LIN {X 0,Y 374.835,Z 474.63,A -85,B 0,C 180,E1 -12336.098,E2 -12336.098} C_VEL
LIN {X 0,Y 375.153,Z 469.967,A -85,B 0,C 180,E1 -12337.535,E2 -12337.535} C_VEL
LIN {X 0,Y 375.66,Z 463.156,A -85,B 0,C 180,E1 -12339.15,E2 -12339.15} C_VEL
LIN {X 0,Y 376.273,Z 455.706,A -85,B 0,C 180,E1 -12340.492,E2 -12340.492} C_VEL
LIN {X 0,Y 376.913,Z 448.357,A -85,B 0,C 180,E1 -12341.563,E2 -12341.563} C_VEL
LIN {X 0,Y 377.501,Z 440.485,A -85,B 0,C 180,E1 -12342.499,E2 -12342.499} C_VEL
LIN {X 0,Y 378.112,Z 432.163,A -85,B 0,C 180,E1 -12343.298,E2 -12343.298} C_VEL
LIN {X 0,Y 378.757,Z 421.529,A -85,B 0,C 180,E1 -12344.095,E2 -12344.095} C_VEL
LIN {X 0,Y 379.284,Z 409.946,A -85,B 0,C 180,E1 -12344.692,E2 -12344.692} C_VEL
LIN {X 0,Y 379.632,Z 400.236,A -85,B 0,C 180,E1 -12345.021,E2 -12345.021} C_VEL
LIN {X 0,Y 380.166,Z 346.091,A -85,B 0,C 180,E1 -12346.072,E2 -12346.072} C_VEL
LIN {X 0,Y 376.584,Z 324.274,A -85,B 0,C 180,E1 -12346.671,E2 -12346.671} C_VEL
LIN {X 0,Y 376.541,Z 323.244,A -85,B 0,C 180,E1 -12346.816,E2 -12346.816} C_VEL
LIN {X 0,Y 377.372,Z 311.444,A -85,B 0,C 180,E1 -12350.153,E2 -12350.153} C_VEL
LIN {X 0,Y 377.425,Z 307.16,A -85,B 0,C 180,E1 -12351.402,E2 -12351.402} C_VEL
LIN {X 0,Y 376.03,Z 298.57,A -85,B 0,C 180,E1 -12354.068,E2 -12354.068} C_VEL
LIN {X 0,Y 375.922,Z 298.47,A -85,B 0,C 180,E1 -12357.864,E2 -12357.864} C_VEL
LIN {X 0,Y 375.953,Z 298.469,A -85,B 0,C 180,E1 -12361.562,E2 -12361.562} C_VEL
LIN {X 0,Y 375.951,Z 298.47,A -85,B 0,C 180,E1 -12365.415,E2 -12365.415} C_VEL
LIN {X 0,Y 375.931,Z 298.466,A -85,B 0,C 180,E1 -12368.262,E2 -12368.262} C_VEL
LIN {X 0,Y 375.908,Z 298.472,A -85,B 0,C 180,E1 -12371.596,E2 -12371.596} C_VEL
LIN {X 0,Y 375.915,Z 298.471,A -85,B 0,C 180,E1 -12374.73,E2 -12374.73} C_VEL
LIN {X 0,Y 375.901,Z 298.471,A -85,B 0,C 180,E1 -12377.696,E2 -12377.696} C_VEL
LIN {X 0,Y 375.928,Z 298.469,A -85,B 0,C 180,E1 -12380.533,E2 -12380.533} C_VEL
LIN {X 0,Y 375.951,Z 298.465,A -85,B 0,C 180,E1 -12383.496,E2 -12383.496} C_VEL
LIN {X 0,Y 375.95,Z 298.464,A -85,B 0,C 180,E1 -12385.888,E2 -12385.888} C_VEL
LIN {X 0,Y 375.953,Z 298.464,A -85,B 0,C 180,E1 -12389.686,E2 -12389.686} C_VEL
LIN {X 0,Y 375.909,Z 298.47,A -85,B 0,C 180,E1 -12392.134,E2 -12392.134} C_VEL
LIN {X 0,Y 375.928,Z 298.472,A -85,B 0,C 180,E1 -12394.533,E2 -12394.533} C_VEL
LIN {X 0,Y 375.962,Z 298.466,A -85,B 0,C 180,E1 -12396.886,E2 -12396.886} C_VEL
LIN {X 0,Y 375.965,Z 298.467,A -85,B 0,C 180,E1 -12400.338,E2 -12400.338} C_VEL
LIN {X 0,Y 375.964,Z 298.463,A -85,B 0,C 180,E1 -12403.716,E2 -12403.716} C_VEL
LIN {X 0,Y 376.094,Z 298.447,A -85,B 0,C 180,E1 -12407.042,E2 -12407.042} C_VEL
LIN {X 0,Y 376.103,Z 298.451,A -85,B 0,C 180,E1 -12410.318,E2 -12410.318} C_VEL
LIN {X 0,Y 376.188,Z 298.435,A -85,B 0,C 180,E1 -12413.564,E2 -12413.564} C_VEL
LIN {X 0,Y 376.327,Z 298.421,A -85,B 0,C 180,E1 -12417.86,E2 -12417.86} C_VEL
LIN {X 0,Y 376.322,Z 298.422,A -85,B 0,C 180,E1 -12422.141,E2 -12422.141} C_VEL
LIN {X 0,Y 376.188,Z 298.436,A -85,B 0,C 180,E1 -12426.436,E2 -12426.436} C_VEL
LIN {X 0,Y 376.097,Z 298.451,A -85,B 0,C 180,E1 -12429.682,E2 -12429.682} C_VEL
LIN {X 0,Y 376.081,Z 298.454,A -85,B 0,C 180,E1 -12433.658,E2 -12433.658} C_VEL
LIN {X 0,Y 375.998,Z 298.465,A -85,B 0,C 180,E1 -12437.589,E2 -12437.589} C_VEL
LIN {X 0,Y 375.971,Z 298.462,A -85,B 0,C 180,E1 -12440.833,E2 -12440.833} C_VEL
LIN {X 0,Y 375.926,Z 298.467,A -85,B 0,C 180,E1 -12444.286,E2 -12444.286} C_VEL
LIN {X 0,Y 375.903,Z 298.47,A -85,B 0,C 180,E1 -12446.661,E2 -12446.661} C_VEL
LIN {X 0,Y 375.906,Z 298.473,A -85,B 0,C 180,E1 -12449.085,E2 -12449.085} C_VEL
LIN {X 0,Y 375.947,Z 298.467,A -85,B 0,C 180,E1 -12451.563,E2 -12451.563} C_VEL
LIN {X 0,Y 375.943,Z 298.469,A -85,B 0,C 180,E1 -12455.417,E2 -12455.417} C_VEL
LIN {X 0,Y 375.929,Z 298.467,A -85,B 0,C 180,E1 -12458.263,E2 -12458.263} C_VEL
LIN {X 0,Y 375.908,Z 298.47,A -85,B 0,C 180,E1 -12461.598,E2 -12461.598} C_VEL
LIN {X 0,Y 375.916,Z 298.472,A -85,B 0,C 180,E1 -12464.731,E2 -12464.731} C_VEL
LIN {X 0,Y 375.903,Z 298.47,A -85,B 0,C 180,E1 -12467.697,E2 -12467.697} C_VEL
LIN {X 0,Y 375.931,Z 298.47,A -85,B 0,C 180,E1 -12470.535,E2 -12470.535} C_VEL
LIN {X 0,Y 375.959,Z 298.463,A -85,B 0,C 180,E1 -12473.497,E2 -12473.497} C_VEL
LIN {X 0,Y 375.956,Z 298.464,A -85,B 0,C 180,E1 -12475.889,E2 -12475.889} C_VEL
LIN {X 0,Y 375.957,Z 298.463,A -85,B 0,C 180,E1 -12479.688,E2 -12479.688} C_VEL
LIN {X 0,Y 375.915,Z 298.471,A -85,B 0,C 180,E1 -12482.136,E2 -12482.136} C_VEL
LIN {X 0,Y 376.046,Z 298.57,A -85,B 0,C 180,E1 -12485.976,E2 -12485.976} C_VEL
LIN {X 0,Y 377.411,Z 307.03,A -85,B 0,C 180,E1 -12488.604,E2 -12488.604} C_VEL
LIN {X 0,Y 377.223,Z 313.241,A -85,B 0,C 180,E1 -12490.406,E2 -12490.406} C_VEL
LIN {X 0,Y 376.539,Z 323.725,A -85,B 0,C 180,E1 -12493.324,E2 -12493.324} C_VEL
LIN {X 0,Y 377.181,Z 328.108,A -85,B 0,C 180,E1 -12493.493,E2 -12493.493} C_VEL
LIN {X 0,Y 380.2,Z 346.979,A -85,B 0,C 180,E1 -12493.992,E2 -12493.992} C_VEL
LIN {X 0,Y 379.651,Z 399.832,A -85,B 0,C 180,E1 -12495.014,E2 -12495.014} C_VEL
LIN {X 0,Y 379.356,Z 408.855,A -85,B 0,C 180,E1 -12495.311,E2 -12495.311} C_VEL
LIN {X 0,Y 378.925,Z 418.416,A -85,B 0,C 180,E1 -12495.774,E2 -12495.774} C_VEL
LIN {X 0,Y 378.378,Z 428.445,A -85,B 0,C 180,E1 -12496.438,E2 -12496.438} C_VEL
LIN {X 0,Y 377.632,Z 438.849,A -85,B 0,C 180,E1 -12497.369,E2 -12497.369} C_VEL
LIN {X 0,Y 377.021,Z 446.999,A -85,B 0,C 180,E1 -12498.304,E2 -12498.304} C_VEL
LIN {X 0,Y 376.473,Z 453.724,A -85,B 0,C 180,E1 -12499.241,E2 -12499.241} C_VEL
LIN {X 0,Y 375.895,Z 460.092,A -85,B 0,C 180,E1 -12500.313,E2 -12500.313} C_VEL
LIN {X 0,Y 375.406,Z 466.559,A -85,B 0,C 180,E1 -12501.658,E2 -12501.658} C_VEL
LIN {X 0,Y 375.086,Z 471.723,A -85,B 0,C 180,E1 -12503.005,E2 -12503.005} C_VEL
LIN {X 0,Y 374.779,Z 476.499,A -85,B 0,C 180,E1 -12504.62,E2 -12504.62} C_VEL
LIN {X 0,Y 374.64,Z 478.829,A -85,B 0,C 180,E1 -12505.697,E2 -12505.697} C_VEL
LIN {X 0,Y 374.492,Z 480.603,A -85,B 0,C 180,E1 -12506.773,E2 -12506.773} C_VEL
LIN {X 0,Y 374.461,Z 481.882,A -85,B 0,C 180,E1 -12507.849,E2 -12507.849} C_VEL
LIN {X 0,Y 374.457,Z 482.69,A -85,B 0,C 180,E1 -12508.925,E2 -12508.925} C_VEL
LIN {X 0,Y 374.44,Z 482.998,A -85,B 0,C 180,E1 -12510,E2 -12510} C_VEL
LIN {X 0,Y 374.454,Z 482.72,A -85,B 0,C 180,E1 -12511.075,E2 -12511.075} C_VEL
LIN {X 0,Y 374.444,Z 481.973,A -85,B 0,C 180,E1 -12512.151,E2 -12512.151} C_VEL
LIN {X 0,Y 374.485,Z 480.755,A -85,B 0,C 180,E1 -12513.227,E2 -12513.227} C_VEL
LIN {X 0,Y 374.707,Z 477.894,A -85,B 0,C 180,E1 -12514.842,E2 -12514.842} C_VEL
LIN {X 0,Y 374.825,Z 474.83,A -85,B 0,C 180,E1 -12516.083,E2 -12516.083} C_VEL
LIN {X 0,Y 375.16,Z 470.167,A -85,B 0,C 180,E1 -12517.535,E2 -12517.535} C_VEL
LIN {X 0,Y 375.545,Z 464.655,A -85,B 0,C 180,E1 -12518.881,E2 -12518.881} C_VEL
LIN {X 0,Y 376.175,Z 457.735,A -85,B 0,C 180,E1 -12520.223,E2 -12520.223} C_VEL
LIN {X 0,Y 376.798,Z 449.79,A -85,B 0,C 180,E1 -12521.43,E2 -12521.43} C_VEL
LIN {X 0,Y 377.376,Z 442.216,A -85,B 0,C 180,E1 -12522.366,E2 -12522.366} C_VEL
LIN {X 0,Y 378.043,Z 434.279,A -85,B 0,C 180,E1 -12523.163,E2 -12523.163} C_VEL
LIN {X 0,Y 378.538,Z 426.084,A -85,B 0,C 180,E1 -12523.83,E2 -12523.83} C_VEL
LIN {X 0,Y 378.982,Z 417.782,A -85,B 0,C 180,E1 -12524.361,E2 -12524.361} C_VEL
LIN {X 0,Y 379.342,Z 408.815,A -85,B 0,C 180,E1 -12524.792,E2 -12524.792} C_VEL
LIN {X 0,Y 379.53,Z 403.476,A -85,B 0,C 180,E1 -12524.995,E2 -12524.995} C_VEL
LIN {X 0,Y 379.115,Z 397.696,A -85,B 0,C 180,E1 -12525.169,E2 -12525.169} C_VEL
LIN {X 0,Y 376.426,Z 388.36,A -85,B 0,C 180,E1 -12525.475,E2 -12525.475} C_VEL
LIN {X 0,Y 373.709,Z 379.004,A -85,B 0,C 180,E1 -12525.772,E2 -12525.772} C_VEL
LIN {X 0,Y 373.119,Z 373.187,A -85,B 0,C 180,E1 -12525.909,E2 -12525.909} C_VEL
LIN {X 0,Y 373.222,Z 346.278,A -85,B 0,C 180,E1 -12526.433,E2 -12526.433} C_VEL
LIN {X 0,Y 369.609,Z 324.06,A -85,B 0,C 180,E1 -12527.07,E2 -12527.07} C_VEL
LIN {X 0,Y 369.646,Z 322.378,A -85,B 0,C 180,E1 -12527.424,E2 -12527.424} C_VEL
LIN {X 0,Y 370.417,Z 311.641,A -85,B 0,C 180,E1 -12530.548,E2 -12530.548} C_VEL
LIN {X 0,Y 370.302,Z 307.197,A -85,B 0,C 180,E1 -12531.882,E2 -12531.882} C_VEL
LIN {X 0,Y 368.991,Z 299.445,A -85,B 0,C 180,E1 -12534.36,E2 -12534.36} C_VEL
LIN {X 0,Y 368.863,Z 299.349,A -85,B 0,C 180,E1 -12537.211,E2 -12537.211} C_VEL
LIN {X 0,Y 368.892,Z 299.348,A -85,B 0,C 180,E1 -12539.692,E2 -12539.692} C_VEL
LIN {X 0,Y 368.894,Z 299.345,A -85,B 0,C 180,E1 -12543.042,E2 -12543.042} C_VEL
LIN {X 0,Y 368.913,Z 299.341,A -85,B 0,C 180,E1 -12546.196,E2 -12546.196} C_VEL
LIN {X 0,Y 368.871,Z 299.349,A -85,B 0,C 180,E1 -12548.956,E2 -12548.956} C_VEL
LIN {X 0,Y 368.854,Z 299.348,A -85,B 0,C 180,E1 -12552.004,E2 -12552.004} C_VEL
LIN {X 0,Y 368.869,Z 299.352,A -85,B 0,C 180,E1 -12555.174,E2 -12555.174} C_VEL
LIN {X 0,Y 368.859,Z 299.347,A -85,B 0,C 180,E1 -12558.174,E2 -12558.174} C_VEL
LIN {X 0,Y 368.872,Z 299.348,A -85,B 0,C 180,E1 -12561.365,E2 -12561.365} C_VEL
LIN {X 0,Y 368.925,Z 299.343,A -85,B 0,C 180,E1 -12565.145,E2 -12565.145} C_VEL
LIN {X 0,Y 368.906,Z 299.345,A -85,B 0,C 180,E1 -12569.044,E2 -12569.044} C_VEL
LIN {X 0,Y 368.9,Z 299.342,A -85,B 0,C 180,E1 -12571.557,E2 -12571.557} C_VEL
LIN {X 0,Y 368.878,Z 299.346,A -85,B 0,C 180,E1 -12575.219,E2 -12575.219} C_VEL
LIN {X 0,Y 368.888,Z 299.344,A -85,B 0,C 180,E1 -12577.602,E2 -12577.602} C_VEL
LIN {X 0,Y 368.905,Z 299.343,A -85,B 0,C 180,E1 -12581.103,E2 -12581.103} C_VEL
LIN {X 0,Y 368.93,Z 299.344,A -85,B 0,C 180,E1 -12584.532,E2 -12584.532} C_VEL
LIN {X 0,Y 369.049,Z 299.326,A -85,B 0,C 180,E1 -12586.79,E2 -12586.79} C_VEL
LIN {X 0,Y 369.054,Z 299.328,A -85,B 0,C 180,E1 -12590.131,E2 -12590.131} C_VEL
LIN {X 0,Y 369.149,Z 299.312,A -85,B 0,C 180,E1 -12593.441,E2 -12593.441} C_VEL
LIN {X 0,Y 369.291,Z 299.297,A -85,B 0,C 180,E1 -12597.819,E2 -12597.819} C_VEL
LIN {X 0,Y 369.285,Z 299.298,A -85,B 0,C 180,E1 -12602.181,E2 -12602.181} C_VEL
LIN {X 0,Y 369.148,Z 299.312,A -85,B 0,C 180,E1 -12606.559,E2 -12606.559} C_VEL
LIN {X 0,Y 369.048,Z 299.329,A -85,B 0,C 180,E1 -12609.869,E2 -12609.869} C_VEL
LIN {X 0,Y 369.029,Z 299.332,A -85,B 0,C 180,E1 -12613.772,E2 -12613.772} C_VEL
LIN {X 0,Y 368.945,Z 299.341,A -85,B 0,C 180,E1 -12617.745,E2 -12617.745} C_VEL
LIN {X 0,Y 368.901,Z 299.346,A -85,B 0,C 180,E1 -12621.221,E2 -12621.221} C_VEL
LIN {X 0,Y 368.899,Z 299.344,A -85,B 0,C 180,E1 -12623.874,E2 -12623.874} C_VEL
LIN {X 0,Y 368.849,Z 299.354,A -85,B 0,C 180,E1 -12627.212,E2 -12627.212} C_VEL
LIN {X 0,Y 368.885,Z 299.346,A -85,B 0,C 180,E1 -12629.693,E2 -12629.693} C_VEL
LIN {X 0,Y 368.889,Z 299.348,A -85,B 0,C 180,E1 -12633.043,E2 -12633.043} C_VEL
LIN {X 0,Y 368.904,Z 299.342,A -85,B 0,C 180,E1 -12636.198,E2 -12636.198} C_VEL
LIN {X 0,Y 368.867,Z 299.352,A -85,B 0,C 180,E1 -12638.958,E2 -12638.958} C_VEL
LIN {X 0,Y 368.852,Z 299.348,A -85,B 0,C 180,E1 -12642.006,E2 -12642.006} C_VEL
LIN {X 0,Y 368.868,Z 299.35,A -85,B 0,C 180,E1 -12645.175,E2 -12645.175} C_VEL
LIN {X 0,Y 368.855,Z 299.349,A -85,B 0,C 180,E1 -12648.175,E2 -12648.175} C_VEL
LIN {X 0,Y 368.871,Z 299.347,A -85,B 0,C 180,E1 -12651.367,E2 -12651.367} C_VEL
LIN {X 0,Y 368.931,Z 299.34,A -85,B 0,C 180,E1 -12655.147,E2 -12655.147} C_VEL
LIN {X 0,Y 368.91,Z 299.343,A -85,B 0,C 180,E1 -12659.045,E2 -12659.045} C_VEL
LIN {X 0,Y 368.904,Z 299.342,A -85,B 0,C 180,E1 -12661.558,E2 -12661.558} C_VEL
LIN {X 0,Y 368.937,Z 299.34,A -85,B 0,C 180,E1 -12665.224,E2 -12665.224} C_VEL
LIN {X 0,Y 368.964,Z 299.455,A -85,B 0,C 180,E1 -12665.699,E2 -12665.699} C_VEL
LIN {X 0,Y 370.297,Z 307.05,A -85,B 0,C 180,E1 -12668.118,E2 -12668.118} C_VEL
LIN {X 0,Y 370.438,Z 311.49,A -85,B 0,C 180,E1 -12669.453,E2 -12669.453} C_VEL
LIN {X 0,Y 369.575,Z 323.615,A -85,B 0,C 180,E1 -12672.929,E2 -12672.929} C_VEL
LIN {X 0,Y 370.085,Z 326.931,A -85,B 0,C 180,E1 -12673.085,E2 -12673.085} C_VEL
LIN {X 0,Y 373.379,Z 347.391,A -85,B 0,C 180,E1 -12673.641,E2 -12673.641} C_VEL
LIN {X 0,Y 372.867,Z 399.709,A -85,B 0,C 180,E1 -12674.674,E2 -12674.674} C_VEL
LIN {X 0,Y 372.455,Z 409.396,A -85,B 0,C 180,E1 -12674.998,E2 -12674.998} C_VEL
LIN {X 0,Y 372.037,Z 419.413,A -85,B 0,C 180,E1 -12675.505,E2 -12675.505} C_VEL
LIN {X 0,Y 371.299,Z 430.789,A -85,B 0,C 180,E1 -12676.314,E2 -12676.314} C_VEL
LIN {X 0,Y 370.649,Z 439.356,A -85,B 0,C 180,E1 -12677.127,E2 -12677.127} C_VEL
LIN {X 0,Y 370.052,Z 447.415,A -85,B 0,C 180,E1 -12678.081,E2 -12678.081} C_VEL
LIN {X 0,Y 369.467,Z 454.071,A -85,B 0,C 180,E1 -12679.035,E2 -12679.035} C_VEL
LIN {X 0,Y 368.886,Z 460.388,A -85,B 0,C 180,E1 -12680.127,E2 -12680.127} C_VEL
LIN {X 0,Y 368.433,Z 465.635,A -85,B 0,C 180,E1 -12681.222,E2 -12681.222} C_VEL
LIN {X 0,Y 368.124,Z 470.009,A -85,B 0,C 180,E1 -12682.32,E2 -12682.32} C_VEL
LIN {X 0,Y 367.734,Z 475.123,A -85,B 0,C 180,E1 -12683.951,E2 -12683.951} C_VEL
LIN {X 0,Y 367.64,Z 477.799,A -85,B 0,C 180,E1 -12685.065,E2 -12685.065} C_VEL
LIN {X 0,Y 367.41,Z 480.688,A -85,B 0,C 180,E1 -12686.71,E2 -12686.71} C_VEL
LIN {X 0,Y 367.362,Z 481.933,A -85,B 0,C 180,E1 -12687.807,E2 -12687.807} C_VEL
LIN {X 0,Y 367.355,Z 482.707,A -85,B 0,C 180,E1 -12688.904,E2 -12688.904} C_VEL
LIN {X 0,Y 367.34,Z 483,A -85,B 0,C 180,E1 -12690,E2 -12690} C_VEL
LIN {X 0,Y 367.355,Z 482.704,A -85,B 0,C 180,E1 -12691.096,E2 -12691.096} C_VEL
LIN {X 0,Y 367.362,Z 481.922,A -85,B 0,C 180,E1 -12692.193,E2 -12692.193} C_VEL
LIN {X 0,Y 367.41,Z 480.67,A -85,B 0,C 180,E1 -12693.29,E2 -12693.29} C_VEL
LIN {X 0,Y 367.633,Z 477.774,A -85,B 0,C 180,E1 -12694.935,E2 -12694.935} C_VEL
LIN {X 0,Y 367.836,Z 473.783,A -85,B 0,C 180,E1 -12696.522,E2 -12696.522} C_VEL
LIN {X 0,Y 368.253,Z 467.925,A -85,B 0,C 180,E1 -12698.229,E2 -12698.229} C_VEL
LIN {X 0,Y 368.767,Z 461.741,A -85,B 0,C 180,E1 -12699.599,E2 -12699.599} C_VEL
LIN {X 0,Y 369.29,Z 455.704,A -85,B 0,C 180,E1 -12700.693,E2 -12700.693} C_VEL
LIN {X 0,Y 369.966,Z 448.354,A -85,B 0,C 180,E1 -12701.783,E2 -12701.783} C_VEL
LIN {X 0,Y 370.567,Z 440.481,A -85,B 0,C 180,E1 -12702.737,E2 -12702.737} C_VEL
LIN {X 0,Y 371.208,Z 432.159,A -85,B 0,C 180,E1 -12703.55,E2 -12703.55} C_VEL
LIN {X 0,Y 371.888,Z 421.524,A -85,B 0,C 180,E1 -12704.361,E2 -12704.361} C_VEL
LIN {X 0,Y 372.437,Z 409.937,A -85,B 0,C 180,E1 -12704.968,E2 -12704.968} C_VEL
LIN {X 0,Y 372.791,Z 400.221,A -85,B 0,C 180,E1 -12705.303,E2 -12705.303} C_VEL
LIN {X 0,Y 373.377,Z 346.955,A -85,B 0,C 180,E1 -12706.355,E2 -12706.355} C_VEL
LIN {X 0,Y 369.632,Z 324.261,A -85,B 0,C 180,E1 -12706.994,E2 -12706.994} C_VEL
LIN {X 0,Y 369.572,Z 323.242,A -85,B 0,C 180,E1 -12707.143,E2 -12707.143} C_VEL
LIN {X 0,Y 370.422,Z 311.442,A -85,B 0,C 180,E1 -12710.548,E2 -12710.548} C_VEL
LIN {X 0,Y 370.291,Z 307.003,A -85,B 0,C 180,E1 -12711.882,E2 -12711.882} C_VEL
LIN {X 0,Y 368.982,Z 299.443,A -85,B 0,C 180,E1 -12714.297,E2 -12714.297} C_VEL
LIN {X 0,Y 368.861,Z 299.35,A -85,B 0,C 180,E1 -12717.211,E2 -12717.211} C_VEL
LIN {X 0,Y 368.891,Z 299.348,A -85,B 0,C 180,E1 -12719.692,E2 -12719.692} C_VEL
LIN {X 0,Y 368.892,Z 299.346,A -85,B 0,C 180,E1 -12723.042,E2 -12723.042} C_VEL
LIN {X 0,Y 368.911,Z 299.341,A -85,B 0,C 180,E1 -12726.196,E2 -12726.196} C_VEL
LIN {X 0,Y 368.869,Z 299.349,A -85,B 0,C 180,E1 -12728.956,E2 -12728.956} C_VEL
LIN {X 0,Y 368.853,Z 299.348,A -85,B 0,C 180,E1 -12732.005,E2 -12732.005} C_VEL
LIN {X 0,Y 368.868,Z 299.352,A -85,B 0,C 180,E1 -12735.174,E2 -12735.174} C_VEL
LIN {X 0,Y 368.854,Z 299.348,A -85,B 0,C 180,E1 -12738.174,E2 -12738.174} C_VEL
LIN {X 0,Y 368.87,Z 299.348,A -85,B 0,C 180,E1 -12741.366,E2 -12741.366} C_VEL
LIN {X 0,Y 368.924,Z 299.343,A -85,B 0,C 180,E1 -12745.145,E2 -12745.145} C_VEL
LIN {X 0,Y 368.906,Z 299.345,A -85,B 0,C 180,E1 -12749.044,E2 -12749.044} C_VEL
LIN {X 0,Y 368.899,Z 299.342,A -85,B 0,C 180,E1 -12751.557,E2 -12751.557} C_VEL
LIN {X 0,Y 368.877,Z 299.346,A -85,B 0,C 180,E1 -12755.219,E2 -12755.219} C_VEL
LIN {X 0,Y 368.888,Z 299.344,A -85,B 0,C 180,E1 -12757.602,E2 -12757.602} C_VEL
LIN {X 0,Y 368.905,Z 299.343,A -85,B 0,C 180,E1 -12761.103,E2 -12761.103} C_VEL
LIN {X 0,Y 368.93,Z 299.343,A -85,B 0,C 180,E1 -12764.532,E2 -12764.532} C_VEL
LIN {X 0,Y 369.049,Z 299.326,A -85,B 0,C 180,E1 -12766.79,E2 -12766.79} C_VEL
LIN {X 0,Y 369.053,Z 299.328,A -85,B 0,C 180,E1 -12770.131,E2 -12770.131} C_VEL
LIN {X 0,Y 369.149,Z 299.312,A -85,B 0,C 180,E1 -12773.441,E2 -12773.441} C_VEL
LIN {X 0,Y 369.291,Z 299.297,A -85,B 0,C 180,E1 -12777.819,E2 -12777.819} C_VEL
LIN {X 0,Y 369.285,Z 299.298,A -85,B 0,C 180,E1 -12782.181,E2 -12782.181} C_VEL
LIN {X 0,Y 369.149,Z 299.312,A -85,B 0,C 180,E1 -12786.559,E2 -12786.559} C_VEL
LIN {X 0,Y 369.048,Z 299.329,A -85,B 0,C 180,E1 -12789.869,E2 -12789.869} C_VEL
LIN {X 0,Y 369.029,Z 299.332,A -85,B 0,C 180,E1 -12793.772,E2 -12793.772} C_VEL
LIN {X 0,Y 368.945,Z 299.341,A -85,B 0,C 180,E1 -12797.745,E2 -12797.745} C_VEL
LIN {X 0,Y 368.901,Z 299.345,A -85,B 0,C 180,E1 -12801.221,E2 -12801.221} C_VEL
LIN {X 0,Y 368.9,Z 299.344,A -85,B 0,C 180,E1 -12803.874,E2 -12803.874} C_VEL
LIN {X 0,Y 368.85,Z 299.353,A -85,B 0,C 180,E1 -12807.213,E2 -12807.213} C_VEL
LIN {X 0,Y 368.885,Z 299.346,A -85,B 0,C 180,E1 -12809.693,E2 -12809.693} C_VEL
LIN {X 0,Y 368.889,Z 299.348,A -85,B 0,C 180,E1 -12813.043,E2 -12813.043} C_VEL
LIN {X 0,Y 368.905,Z 299.342,A -85,B 0,C 180,E1 -12816.198,E2 -12816.198} C_VEL
LIN {X 0,Y 368.868,Z 299.351,A -85,B 0,C 180,E1 -12818.958,E2 -12818.958} C_VEL
LIN {X 0,Y 368.853,Z 299.348,A -85,B 0,C 180,E1 -12822.006,E2 -12822.006} C_VEL
LIN {X 0,Y 368.869,Z 299.35,A -85,B 0,C 180,E1 -12825.175,E2 -12825.175} C_VEL
LIN {X 0,Y 368.856,Z 299.348,A -85,B 0,C 180,E1 -12828.175,E2 -12828.175} C_VEL
LIN {X 0,Y 368.873,Z 299.347,A -85,B 0,C 180,E1 -12831.367,E2 -12831.367} C_VEL
LIN {X 0,Y 368.933,Z 299.34,A -85,B 0,C 180,E1 -12835.147,E2 -12835.147} C_VEL
LIN {X 0,Y 368.894,Z 299.345,A -85,B 0,C 180,E1 -12839.044,E2 -12839.044} C_VEL
LIN {X 0,Y 368.905,Z 299.342,A -85,B 0,C 180,E1 -12841.558,E2 -12841.558} C_VEL
LIN {X 0,Y 368.935,Z 299.342,A -85,B 0,C 180,E1 -12845.224,E2 -12845.224} C_VEL
LIN {X 0,Y 369.008,Z 299.593,A -85,B 0,C 180,E1 -12845.826,E2 -12845.826} C_VEL
LIN {X 0,Y 370.38,Z 307.778,A -85,B 0,C 180,E1 -12848.401,E2 -12848.401} C_VEL
LIN {X 0,Y 370.311,Z 313.243,A -85,B 0,C 180,E1 -12850.025,E2 -12850.025} C_VEL
LIN {X 0,Y 369.576,Z 323.586,A -85,B 0,C 180,E1 -12852.975,E2 -12852.975} C_VEL
LIN {X 0,Y 369.703,Z 324.949,A -85,B 0,C 180,E1 -12853.077,E2 -12853.077} C_VEL
LIN {X 0,Y 373.378,Z 347.27,A -85,B 0,C 180,E1 -12853.696,E2 -12853.696} C_VEL
LIN {X 0,Y 372.808,Z 399.85,A -85,B 0,C 180,E1 -12854.732,E2 -12854.732} C_VEL
LIN {X 0,Y 372.506,Z 408.867,A -85,B 0,C 180,E1 -12855.035,E2 -12855.035} C_VEL
LIN {X 0,Y 372.064,Z 418.425,A -85,B 0,C 180,E1 -12855.506,E2 -12855.506} C_VEL
LIN {X 0,Y 371.49,Z 428.452,A -85,B 0,C 180,E1 -12856.182,E2 -12856.182} C_VEL
LIN {X 0,Y 370.7,Z 438.854,A -85,B 0,C 180,E1 -12857.129,E2 -12857.129} C_VEL
LIN {X 0,Y 370.068,Z 447.003,A -85,B 0,C 180,E1 -12858.081,E2 -12858.081} C_VEL
LIN {X 0,Y 369.486,Z 453.727,A -85,B 0,C 180,E1 -12859.035,E2 -12859.035} C_VEL
LIN {X 0,Y 368.895,Z 460.094,A -85,B 0,C 180,E1 -12860.127,E2 -12860.127} C_VEL
LIN {X 0,Y 368.385,Z 466.562,A -85,B 0,C 180,E1 -12861.498,E2 -12861.498} C_VEL
LIN {X 0,Y 368.041,Z 471.722,A -85,B 0,C 180,E1 -12862.87,E2 -12862.87} C_VEL
LIN {X 0,Y 367.688,Z 476.5,A -85,B 0,C 180,E1 -12864.516,E2 -12864.516} C_VEL
LIN {X 0,Y 367.577,Z 478.83,A -85,B 0,C 180,E1 -12865.614,E2 -12865.614} C_VEL
LIN {X 0,Y 367.412,Z 480.604,A -85,B 0,C 180,E1 -12866.71,E2 -12866.71} C_VEL
LIN {X 0,Y 367.363,Z 481.883,A -85,B 0,C 180,E1 -12867.807,E2 -12867.807} C_VEL
LIN {X 0,Y 367.356,Z 482.69,A -85,B 0,C 180,E1 -12868.904,E2 -12868.904} C_VEL
LIN {X 0,Y 367.341,Z 482.998,A -85,B 0,C 180,E1 -12870,E2 -12870} C_VEL
LIN {X 0,Y 367.353,Z 482.72,A -85,B 0,C 180,E1 -12871.096,E2 -12871.096} C_VEL
LIN {X 0,Y 367.347,Z 481.973,A -85,B 0,C 180,E1 -12872.193,E2 -12872.193} C_VEL
LIN {X 0,Y 367.405,Z 480.755,A -85,B 0,C 180,E1 -12873.29,E2 -12873.29} C_VEL
LIN {X 0,Y 367.629,Z 477.893,A -85,B 0,C 180,E1 -12874.935,E2 -12874.935} C_VEL
LIN {X 0,Y 367.831,Z 473.962,A -85,B 0,C 180,E1 -12876.514,E2 -12876.514} C_VEL
LIN {X 0,Y 368.247,Z 468.168,A -85,B 0,C 180,E1 -12878.229,E2 -12878.229} C_VEL
LIN {X 0,Y 368.767,Z 462.037,A -85,B 0,C 180,E1 -12879.599,E2 -12879.599} C_VEL
LIN {X 0,Y 369.301,Z 456.051,A -85,B 0,C 180,E1 -12880.693,E2 -12880.693} C_VEL
LIN {X 0,Y 369.914,Z 448.766,A -85,B 0,C 180,E1 -12881.785,E2 -12881.785} C_VEL
LIN {X 0,Y 370.52,Z 440.982,A -85,B 0,C 180,E1 -12882.738,E2 -12882.738} C_VEL
LIN {X 0,Y 371.239,Z 432.773,A -85,B 0,C 180,E1 -12883.548,E2 -12883.548} C_VEL
LIN {X 0,Y 371.775,Z 424.204,A -85,B 0,C 180,E1 -12884.226,E2 -12884.226} C_VEL
LIN {X 0,Y 372.372,Z 412.86,A -85,B 0,C 180,E1 -12884.901,E2 -12884.901} C_VEL
LIN {X 0,Y 372.762,Z 401.287,A -85,B 0,C 180,E1 -12885.333,E2 -12885.333} C_VEL
LIN {X 0,Y 373.119,Z 373.187,A -85,B 0,C 180,E1 -12885.909,E2 -12885.909} C_VEL
LIN {X 0,Y 372.608,Z 367.369,A -85,B 0,C 180,E1 -12886.046,E2 -12886.046} C_VEL
LIN {X 0,Y 370.067,Z 357.998,A -85,B 0,C 180,E1 -12886.344,E2 -12886.344} C_VEL
LIN {X 0,Y 366.559,Z 346.793,A -85,B 0,C 180,E1 -12886.729,E2 -12886.729} C_VEL
LIN {X 0,Y 365.808,Z 342.941,A -85,B 0,C 180,E1 -12886.842,E2 -12886.842} C_VEL
LIN {X 0,Y 362.669,Z 324.052,A -85,B 0,C 180,E1 -12887.407,E2 -12887.407} C_VEL
LIN {X 0,Y 362.693,Z 322.376,A -85,B 0,C 180,E1 -12887.769,E2 -12887.769} C_VEL
LIN {X 0,Y 363.472,Z 311.639,A -85,B 0,C 180,E1 -12890.959,E2 -12890.959} C_VEL
LIN {X 0,Y 363.19,Z 307.567,A -85,B 0,C 180,E1 -12892.22,E2 -12892.22} C_VEL
LIN {X 0,Y 361.939,Z 300.324,A -85,B 0,C 180,E1 -12894.59,E2 -12894.59} C_VEL
LIN {X 0,Y 361.838,Z 300.226,A -85,B 0,C 180,E1 -12897.784,E2 -12897.784} C_VEL
LIN {X 0,Y 361.845,Z 300.225,A -85,B 0,C 180,E1 -12901.285,E2 -12901.285} C_VEL
LIN {X 0,Y 361.851,Z 300.22,A -85,B 0,C 180,E1 -12904.28,E2 -12904.28} C_VEL
LIN {X 0,Y 361.857,Z 300.225,A -85,B 0,C 180,E1 -12907.221,E2 -12907.221} C_VEL
LIN {X 0,Y 361.806,Z 300.227,A -85,B 0,C 180,E1 -12910.75,E2 -12910.75} C_VEL
LIN {X 0,Y 361.807,Z 300.226,A -85,B 0,C 180,E1 -12914.369,E2 -12914.369} C_VEL
LIN {X 0,Y 361.821,Z 300.226,A -85,B 0,C 180,E1 -12917.569,E2 -12917.569} C_VEL
LIN {X 0,Y 361.838,Z 300.223,A -85,B 0,C 180,E1 -12921.571,E2 -12921.571} C_VEL
LIN {X 0,Y 361.864,Z 300.222,A -85,B 0,C 180,E1 -12924.656,E2 -12924.656} C_VEL
LIN {X 0,Y 361.831,Z 300.225,A -85,B 0,C 180,E1 -12928.37,E2 -12928.37} C_VEL
LIN {X 0,Y 361.86,Z 300.223,A -85,B 0,C 180,E1 -12930.952,E2 -12930.952} C_VEL
LIN {X 0,Y 361.852,Z 300.226,A -85,B 0,C 180,E1 -12934.704,E2 -12934.704} C_VEL
LIN {X 0,Y 361.846,Z 300.225,A -85,B 0,C 180,E1 -12938.344,E2 -12938.344} C_VEL
LIN {X 0,Y 361.896,Z 300.217,A -85,B 0,C 180,E1 -12942.092,E2 -12942.092} C_VEL
LIN {X 0,Y 361.972,Z 300.209,A -85,B 0,C 180,E1 -12946.113,E2 -12946.113} C_VEL
LIN {X 0,Y 361.991,Z 300.206,A -85,B 0,C 180,E1 -12949.937,E2 -12949.937} C_VEL
LIN {X 0,Y 362.112,Z 300.188,A -85,B 0,C 180,E1 -12953.313,E2 -12953.313} C_VEL
LIN {X 0,Y 362.254,Z 300.173,A -85,B 0,C 180,E1 -12957.776,E2 -12957.776} C_VEL
LIN {X 0,Y 362.163,Z 300.182,A -85,B 0,C 180,E1 -12961.112,E2 -12961.112} C_VEL
LIN {X 0,Y 362.248,Z 300.174,A -85,B 0,C 180,E1 -12962.224,E2 -12962.224} C_VEL
LIN {X 0,Y 362.112,Z 300.188,A -85,B 0,C 180,E1 -12966.687,E2 -12966.687} C_VEL
LIN {X 0,Y 361.985,Z 300.207,A -85,B 0,C 180,E1 -12970.063,E2 -12970.063} C_VEL
LIN {X 0,Y 361.971,Z 300.209,A -85,B 0,C 180,E1 -12973.886,E2 -12973.886} C_VEL
LIN {X 0,Y 361.878,Z 300.218,A -85,B 0,C 180,E1 -12978.103,E2 -12978.103} C_VEL
LIN {X 0,Y 361.845,Z 300.226,A -85,B 0,C 180,E1 -12981.656,E2 -12981.656} C_VEL
LIN {X 0,Y 361.852,Z 300.226,A -85,B 0,C 180,E1 -12985.296,E2 -12985.296} C_VEL
LIN {X 0,Y 361.848,Z 300.225,A -85,B 0,C 180,E1 -12989.074,E2 -12989.074} C_VEL
LIN {X 0,Y 361.84,Z 300.225,A -85,B 0,C 180,E1 -12992.945,E2 -12992.945} C_VEL
LIN {X 0,Y 361.857,Z 300.221,A -85,B 0,C 180,E1 -12995.638,E2 -12995.638} C_VEL
LIN {X 0,Y 361.819,Z 300.23,A -85,B 0,C 180,E1 -12999.018,E2 -12999.018} C_VEL
LIN {X 0,Y 361.823,Z 300.229,A -85,B 0,C 180,E1 -13002.831,E2 -13002.831} C_VEL
LIN {X 0,Y 361.807,Z 300.226,A -85,B 0,C 180,E1 -13005.948,E2 -13005.948} C_VEL
LIN {X 0,Y 361.805,Z 300.228,A -85,B 0,C 180,E1 -13009.25,E2 -13009.25} C_VEL
LIN {X 0,Y 361.859,Z 300.223,A -85,B 0,C 180,E1 -13012.982,E2 -13012.982} C_VEL
LIN {X 0,Y 361.854,Z 300.226,A -85,B 0,C 180,E1 -13016.632,E2 -13016.632} C_VEL
LIN {X 0,Y 361.852,Z 300.22,A -85,B 0,C 180,E1 -13019.671,E2 -13019.671} C_VEL
LIN {X 0,Y 361.852,Z 300.22,A -85,B 0,C 180,E1 -13023.468,E2 -13023.468} C_VEL
LIN {X 0,Y 361.921,Z 300.383,A -85,B 0,C 180,E1 -13025.492,E2 -13025.492} C_VEL
LIN {X 0,Y 363.371,Z 308.696,A -85,B 0,C 180,E1 -13028.183,E2 -13028.183} C_VEL
LIN {X 0,Y 363.378,Z 313.443,A -85,B 0,C 180,E1 -13029.627,E2 -13029.627} C_VEL
LIN {X 0,Y 362.638,Z 323.618,A -85,B 0,C 180,E1 -13032.592,E2 -13032.592} C_VEL
LIN {X 0,Y 363.158,Z 326.951,A -85,B 0,C 180,E1 -13032.753,E2 -13032.753} C_VEL
LIN {X 0,Y 366.556,Z 347.643,A -85,B 0,C 180,E1 -13033.333,E2 -13033.333} C_VEL
LIN {X 0,Y 366.032,Z 399.773,A -85,B 0,C 180,E1 -13034.382,E2 -13034.382} C_VEL
LIN {X 0,Y 365.625,Z 409.405,A -85,B 0,C 180,E1 -13034.711,E2 -13034.711} C_VEL
LIN {X 0,Y 365.174,Z 419.42,A -85,B 0,C 180,E1 -13035.226,E2 -13035.226} C_VEL
LIN {X 0,Y 364.423,Z 430.793,A -85,B 0,C 180,E1 -13036.051,E2 -13036.051} C_VEL
LIN {X 0,Y 363.748,Z 439.36,A -85,B 0,C 180,E1 -13036.878,E2 -13036.878} C_VEL
LIN {X 0,Y 363.111,Z 447.418,A -85,B 0,C 180,E1 -13037.85,E2 -13037.85} C_VEL
LIN {X 0,Y 362.484,Z 454.074,A -85,B 0,C 180,E1 -13038.821,E2 -13038.821} C_VEL
LIN {X 0,Y 361.902,Z 460.39,A -85,B 0,C 180,E1 -13039.935,E2 -13039.935} C_VEL
LIN {X 0,Y 361.411,Z 465.636,A -85,B 0,C 180,E1 -13041.05,E2 -13041.05} C_VEL
LIN {X 0,Y 361.067,Z 470.011,A -85,B 0,C 180,E1 -13042.169,E2 -13042.169} C_VEL
LIN {X 0,Y 360.72,Z 474.325,A -85,B 0,C 180,E1 -13043.537,E2 -13043.537} C_VEL
LIN {X 0,Y 360.564,Z 477.8,A -85,B 0,C 180,E1 -13044.968,E2 -13044.968} C_VEL
LIN {X 0,Y 360.333,Z 480.689,A -85,B 0,C 180,E1 -13046.646,E2 -13046.646} C_VEL
LIN {X 0,Y 360.268,Z 481.933,A -85,B 0,C 180,E1 -13047.764,E2 -13047.764} C_VEL
LIN {X 0,Y 360.255,Z 482.707,A -85,B 0,C 180,E1 -13048.882,E2 -13048.882} C_VEL
LIN {X 0,Y 360.24,Z 483,A -85,B 0,C 180,E1 -13050,E2 -13050} C_VEL
LIN {X 0,Y 360.255,Z 482.703,A -85,B 0,C 180,E1 -13051.118,E2 -13051.118} C_VEL
LIN {X 0,Y 360.268,Z 481.922,A -85,B 0,C 180,E1 -13052.236,E2 -13052.236} C_VEL
LIN {X 0,Y 360.333,Z 480.67,A -85,B 0,C 180,E1 -13053.354,E2 -13053.354} C_VEL
LIN {X 0,Y 360.557,Z 477.773,A -85,B 0,C 180,E1 -13055.032,E2 -13055.032} C_VEL
LIN {X 0,Y 360.756,Z 474.151,A -85,B 0,C 180,E1 -13056.514,E2 -13056.514} C_VEL
LIN {X 0,Y 361.127,Z 469.006,A -85,B 0,C 180,E1 -13058.111,E2 -13058.111} C_VEL
LIN {X 0,Y 361.625,Z 463.152,A -85,B 0,C 180,E1 -13059.508,E2 -13059.508} C_VEL
LIN {X 0,Y 362.315,Z 455.701,A -85,B 0,C 180,E1 -13060.901,E2 -13060.901} C_VEL
LIN {X 0,Y 363.028,Z 448.351,A -85,B 0,C 180,E1 -13062.012,E2 -13062.012} C_VEL
LIN {X 0,Y 363.631,Z 440.478,A -85,B 0,C 180,E1 -13062.984,E2 -13062.984} C_VEL
LIN {X 0,Y 364.294,Z 432.154,A -85,B 0,C 180,E1 -13063.812,E2 -13063.812} C_VEL
LIN {X 0,Y 365.024,Z 421.518,A -85,B 0,C 180,E1 -13064.637,E2 -13064.637} C_VEL
LIN {X 0,Y 365.595,Z 409.927,A -85,B 0,C 180,E1 -13065.255,E2 -13065.255} C_VEL
LIN {X 0,Y 365.958,Z 400.207,A -85,B 0,C 180,E1 -13065.596,E2 -13065.596} C_VEL
LIN {X 0,Y 366.508,Z 347.304,A -85,B 0,C 180,E1 -13066.663,E2 -13066.663} C_VEL
LIN {X 0,Y 362.657,Z 324.242,A -85,B 0,C 180,E1 -13067.332,E2 -13067.332} C_VEL
LIN {X 0,Y 362.635,Z 323.241,A -85,B 0,C 180,E1 -13067.481,E2 -13067.481} C_VEL
LIN {X 0,Y 363.367,Z 313.393,A -85,B 0,C 180,E1 -13070.373,E2 -13070.373} C_VEL
LIN {X 0,Y 363.367,Z 308.65,A -85,B 0,C 180,E1 -13071.816,E2 -13071.816} C_VEL
LIN {X 0,Y 361.906,Z 300.314,A -85,B 0,C 180,E1 -13074.551,E2 -13074.551} C_VEL
LIN {X 0,Y 361.837,Z 300.226,A -85,B 0,C 180,E1 -13077.784,E2 -13077.784} C_VEL
LIN {X 0,Y 361.844,Z 300.226,A -85,B 0,C 180,E1 -13081.285,E2 -13081.285} C_VEL
LIN {X 0,Y 361.85,Z 300.221,A -85,B 0,C 180,E1 -13084.28,E2 -13084.28} C_VEL
LIN {X 0,Y 361.855,Z 300.225,A -85,B 0,C 180,E1 -13087.221,E2 -13087.221} C_VEL
LIN {X 0,Y 361.805,Z 300.228,A -85,B 0,C 180,E1 -13090.75,E2 -13090.75} C_VEL
LIN {X 0,Y 361.806,Z 300.226,A -85,B 0,C 180,E1 -13094.369,E2 -13094.369} C_VEL
LIN {X 0,Y 361.816,Z 300.226,A -85,B 0,C 180,E1 -13097.57,E2 -13097.57} C_VEL
LIN {X 0,Y 361.836,Z 300.223,A -85,B 0,C 180,E1 -13101.571,E2 -13101.571} C_VEL
LIN {X 0,Y 361.863,Z 300.223,A -85,B 0,C 180,E1 -13104.656,E2 -13104.656} C_VEL
LIN {X 0,Y 361.83,Z 300.225,A -85,B 0,C 180,E1 -13108.37,E2 -13108.37} C_VEL
LIN {X 0,Y 361.859,Z 300.223,A -85,B 0,C 180,E1 -13110.952,E2 -13110.952} C_VEL
LIN {X 0,Y 361.852,Z 300.226,A -85,B 0,C 180,E1 -13114.704,E2 -13114.704} C_VEL
LIN {X 0,Y 361.845,Z 300.225,A -85,B 0,C 180,E1 -13118.344,E2 -13118.344} C_VEL
LIN {X 0,Y 361.896,Z 300.217,A -85,B 0,C 180,E1 -13122.093,E2 -13122.093} C_VEL
LIN {X 0,Y 361.971,Z 300.209,A -85,B 0,C 180,E1 -13126.113,E2 -13126.113} C_VEL
LIN {X 0,Y 361.99,Z 300.206,A -85,B 0,C 180,E1 -13129.937,E2 -13129.937} C_VEL
LIN {X 0,Y 362.112,Z 300.188,A -85,B 0,C 180,E1 -13133.313,E2 -13133.313} C_VEL
LIN {X 0,Y 362.254,Z 300.173,A -85,B 0,C 180,E1 -13137.776,E2 -13137.776} C_VEL
LIN {X 0,Y 362.163,Z 300.181,A -85,B 0,C 180,E1 -13141.112,E2 -13141.112} C_VEL
LIN {X 0,Y 362.248,Z 300.174,A -85,B 0,C 180,E1 -13142.224,E2 -13142.224} C_VEL
LIN {X 0,Y 362.112,Z 300.188,A -85,B 0,C 180,E1 -13146.687,E2 -13146.687} C_VEL
LIN {X 0,Y 361.985,Z 300.207,A -85,B 0,C 180,E1 -13150.063,E2 -13150.063} C_VEL
LIN {X 0,Y 361.971,Z 300.209,A -85,B 0,C 180,E1 -13153.887,E2 -13153.887} C_VEL
LIN {X 0,Y 361.878,Z 300.218,A -85,B 0,C 180,E1 -13158.104,E2 -13158.104} C_VEL
LIN {X 0,Y 361.845,Z 300.226,A -85,B 0,C 180,E1 -13161.656,E2 -13161.656} C_VEL
LIN {X 0,Y 361.844,Z 300.226,A -85,B 0,C 180,E1 -13165.296,E2 -13165.296} C_VEL
LIN {X 0,Y 361.849,Z 300.224,A -85,B 0,C 180,E1 -13169.074,E2 -13169.074} C_VEL
LIN {X 0,Y 361.84,Z 300.225,A -85,B 0,C 180,E1 -13172.946,E2 -13172.946} C_VEL
LIN {X 0,Y 361.858,Z 300.221,A -85,B 0,C 180,E1 -13175.638,E2 -13175.638} C_VEL
LIN {X 0,Y 361.82,Z 300.23,A -85,B 0,C 180,E1 -13179.019,E2 -13179.019} C_VEL
LIN {X 0,Y 361.824,Z 300.228,A -85,B 0,C 180,E1 -13182.831,E2 -13182.831} C_VEL
LIN {X 0,Y 361.809,Z 300.226,A -85,B 0,C 180,E1 -13185.948,E2 -13185.948} C_VEL
LIN {X 0,Y 361.806,Z 300.228,A -85,B 0,C 180,E1 -13189.25,E2 -13189.25} C_VEL
LIN {X 0,Y 361.86,Z 300.223,A -85,B 0,C 180,E1 -13192.982,E2 -13192.982} C_VEL
LIN {X 0,Y 361.855,Z 300.226,A -85,B 0,C 180,E1 -13196.632,E2 -13196.632} C_VEL
LIN {X 0,Y 361.845,Z 300.221,A -85,B 0,C 180,E1 -13199.67,E2 -13199.67} C_VEL
LIN {X 0,Y 361.853,Z 300.22,A -85,B 0,C 180,E1 -13203.468,E2 -13203.468} C_VEL
LIN {X 0,Y 361.948,Z 300.428,A -85,B 0,C 180,E1 -13205.578,E2 -13205.578} C_VEL
LIN {X 0,Y 363.354,Z 308.524,A -85,B 0,C 180,E1 -13208.19,E2 -13208.19} C_VEL
LIN {X 0,Y 363.374,Z 313.245,A -85,B 0,C 180,E1 -13209.627,E2 -13209.627} C_VEL
LIN {X 0,Y 362.63,Z 323.699,A -85,B 0,C 180,E1 -13212.659,E2 -13212.659} C_VEL
LIN {X 0,Y 363.228,Z 327.468,A -85,B 0,C 180,E1 -13212.826,E2 -13212.826} C_VEL
LIN {X 0,Y 366.599,Z 348.539,A -85,B 0,C 180,E1 -13213.411,E2 -13213.411} C_VEL
LIN {X 0,Y 365.974,Z 399.869,A -85,B 0,C 180,E1 -13214.44,E2 -13214.44} C_VEL
LIN {X 0,Y 365.67,Z 408.878,A -85,B 0,C 180,E1 -13214.748,E2 -13214.748} C_VEL
LIN {X 0,Y 365.198,Z 418.434,A -85,B 0,C 180,E1 -13215.228,E2 -13215.228} C_VEL
LIN {X 0,Y 364.614,Z 428.458,A -85,B 0,C 180,E1 -13215.916,E2 -13215.916} C_VEL
LIN {X 0,Y 363.793,Z 438.858,A -85,B 0,C 180,E1 -13216.88,E2 -13216.88} C_VEL
LIN {X 0,Y 363.122,Z 447.006,A -85,B 0,C 180,E1 -13217.85,E2 -13217.85} C_VEL
LIN {X 0,Y 362.509,Z 453.73,A -85,B 0,C 180,E1 -13218.821,E2 -13218.821} C_VEL
LIN {X 0,Y 361.908,Z 460.097,A -85,B 0,C 180,E1 -13219.935,E2 -13219.935} C_VEL
LIN {X 0,Y 361.448,Z 465.391,A -85,B 0,C 180,E1 -13221.051,E2 -13221.051} C_VEL
LIN {X 0,Y 361.08,Z 469.812,A -85,B 0,C 180,E1 -13222.169,E2 -13222.169} C_VEL
LIN {X 0,Y 360.759,Z 474.026,A -85,B 0,C 180,E1 -13223.485,E2 -13223.485} C_VEL
LIN {X 0,Y 360.566,Z 477.681,A -85,B 0,C 180,E1 -13224.968,E2 -13224.968} C_VEL
LIN {X 0,Y 360.335,Z 480.605,A -85,B 0,C 180,E1 -13226.646,E2 -13226.646} C_VEL
LIN {X 0,Y 360.269,Z 481.883,A -85,B 0,C 180,E1 -13227.764,E2 -13227.764} C_VEL
LIN {X 0,Y 360.256,Z 482.691,A -85,B 0,C 180,E1 -13228.882,E2 -13228.882} C_VEL
LIN {X 0,Y 360.242,Z 482.998,A -85,B 0,C 180,E1 -13230,E2 -13230} C_VEL
LIN {X 0,Y 360.252,Z 482.72,A -85,B 0,C 180,E1 -13231.118,E2 -13231.118} C_VEL
LIN {X 0,Y 360.253,Z 481.972,A -85,B 0,C 180,E1 -13232.236,E2 -13232.236} C_VEL
LIN {X 0,Y 360.329,Z 480.754,A -85,B 0,C 180,E1 -13233.354,E2 -13233.354} C_VEL
LIN {X 0,Y 360.552,Z 477.892,A -85,B 0,C 180,E1 -13235.032,E2 -13235.032} C_VEL
LIN {X 0,Y 360.716,Z 474.468,A -85,B 0,C 180,E1 -13236.455,E2 -13236.455} C_VEL
LIN {X 0,Y 361.058,Z 470.163,A -85,B 0,C 180,E1 -13237.831,E2 -13237.831} C_VEL
LIN {X 0,Y 361.508,Z 464.651,A -85,B 0,C 180,E1 -13239.229,E2 -13239.229} C_VEL
LIN {X 0,Y 362.164,Z 457.73,A -85,B 0,C 180,E1 -13240.623,E2 -13240.623} C_VEL
LIN {X 0,Y 362.883,Z 449.783,A -85,B 0,C 180,E1 -13241.875,E2 -13241.875} C_VEL
LIN {X 0,Y 363.522,Z 442.207,A -85,B 0,C 180,E1 -13242.846,E2 -13242.846} C_VEL
LIN {X 0,Y 364.252,Z 434.268,A -85,B 0,C 180,E1 -13243.671,E2 -13243.671} C_VEL
LIN {X 0,Y 364.791,Z 426.07,A -85,B 0,C 180,E1 -13244.362,E2 -13244.362} C_VEL
LIN {X 0,Y 365.267,Z 417.765,A -85,B 0,C 180,E1 -13244.912,E2 -13244.912} C_VEL
LIN {X 0,Y 365.65,Z 408.791,A -85,B 0,C 180,E1 -13245.36,E2 -13245.36} C_VEL
LIN {X 0,Y 366.014,Z 399.295,A -85,B 0,C 180,E1 -13245.677,E2 -13245.677} C_VEL
LIN {X 0,Y 366.505,Z 347.579,A -85,B 0,C 180,E1 -13246.716,E2 -13246.716} C_VEL
LIN {X 0,Y 365.808,Z 342.941,A -85,B 0,C 180,E1 -13246.842,E2 -13246.842} C_VEL
LIN {X 0,Y 364.61,Z 339.242,A -85,B 0,C 180,E1 -13246.977,E2 -13246.977} C_VEL
LIN {X 0,Y 360.954,Z 333.863,A -85,B 0,C 180,E1 -13247.26,E2 -13247.26} C_VEL
LIN {X 0,Y 357.198,Z 328.544,A -85,B 0,C 180,E1 -13247.557,E2 -13247.557} C_VEL
LIN {X 0,Y 355.845,Z 324.931,A -85,B 0,C 180,E1 -13247.712,E2 -13247.712} C_VEL
LIN {X 0,Y 355.696,Z 323.476,A -85,B 0,C 180,E1 -13247.833,E2 -13247.833} C_VEL
LIN {X 0,Y 356.449,Z 313.589,A -85,B 0,C 180,E1 -13250.787,E2 -13250.787} C_VEL
LIN {X 0,Y 356.337,Z 309.608,A -85,B 0,C 180,E1 -13252.031,E2 -13252.031} C_VEL
LIN {X 0,Y 354.882,Z 301.196,A -85,B 0,C 180,E1 -13254.847,E2 -13254.847} C_VEL
LIN {X 0,Y 354.797,Z 301.099,A -85,B 0,C 180,E1 -13258.385,E2 -13258.385} C_VEL
LIN {X 0,Y 354.785,Z 301.101,A -85,B 0,C 180,E1 -13262.333,E2 -13262.333} C_VEL
LIN {X 0,Y 354.818,Z 301.099,A -85,B 0,C 180,E1 -13265.698,E2 -13265.698} C_VEL
LIN {X 0,Y 354.765,Z 301.107,A -85,B 0,C 180,E1 -13269.412,E2 -13269.412} C_VEL
LIN {X 0,Y 354.777,Z 301.103,A -85,B 0,C 180,E1 -13272.865,E2 -13272.865} C_VEL
LIN {X 0,Y 354.758,Z 301.104,A -85,B 0,C 180,E1 -13276.102,E2 -13276.102} C_VEL
LIN {X 0,Y 354.759,Z 301.107,A -85,B 0,C 180,E1 -13279.175,E2 -13279.175} C_VEL
LIN {X 0,Y 354.794,Z 301.099,A -85,B 0,C 180,E1 -13282.404,E2 -13282.404} C_VEL
LIN {X 0,Y 354.802,Z 301.104,A -85,B 0,C 180,E1 -13284.94,E2 -13284.94} C_VEL
LIN {X 0,Y 354.787,Z 301.103,A -85,B 0,C 180,E1 -13288.405,E2 -13288.405} C_VEL
LIN {X 0,Y 354.79,Z 301.1,A -85,B 0,C 180,E1 -13291.614,E2 -13291.614} C_VEL
LIN {X 0,Y 354.797,Z 301.099,A -85,B 0,C 180,E1 -13295.419,E2 -13295.419} C_VEL
LIN {X 0,Y 354.813,Z 301.098,A -85,B 0,C 180,E1 -13299.112,E2 -13299.112} C_VEL
LIN {X 0,Y 354.843,Z 301.097,A -85,B 0,C 180,E1 -13302.717,E2 -13302.717} C_VEL
LIN {X 0,Y 354.931,Z 301.087,A -85,B 0,C 180,E1 -13306.254,E2 -13306.254} C_VEL
LIN {X 0,Y 354.947,Z 301.082,A -85,B 0,C 180,E1 -13309.735,E2 -13309.735} C_VEL
LIN {X 0,Y 355.078,Z 301.064,A -85,B 0,C 180,E1 -13313.18,E2 -13313.18} C_VEL
LIN {X 0,Y 355.216,Z 301.049,A -85,B 0,C 180,E1 -13317.732,E2 -13317.732} C_VEL
LIN {X 0,Y 355.135,Z 301.057,A -85,B 0,C 180,E1 -13321.134,E2 -13321.134} C_VEL
LIN {X 0,Y 355.21,Z 301.05,A -85,B 0,C 180,E1 -13322.268,E2 -13322.268} C_VEL
LIN {X 0,Y 355.078,Z 301.064,A -85,B 0,C 180,E1 -13326.82,E2 -13326.82} C_VEL
LIN {X 0,Y 354.941,Z 301.083,A -85,B 0,C 180,E1 -13330.265,E2 -13330.265} C_VEL
LIN {X 0,Y 354.914,Z 301.087,A -85,B 0,C 180,E1 -13334.005,E2 -13334.005} C_VEL
LIN {X 0,Y 354.836,Z 301.096,A -85,B 0,C 180,E1 -13338.069,E2 -13338.069} C_VEL
LIN {X 0,Y 354.797,Z 301.099,A -85,B 0,C 180,E1 -13342.108,E2 -13342.108} C_VEL
LIN {X 0,Y 354.791,Z 301.102,A -85,B 0,C 180,E1 -13345.836,E2 -13345.836} C_VEL
LIN {X 0,Y 354.789,Z 301.102,A -85,B 0,C 180,E1 -13349.684,E2 -13349.684} C_VEL
LIN {X 0,Y 354.779,Z 301.101,A -85,B 0,C 180,E1 -13352.334,E2 -13352.334} C_VEL
LIN {X 0,Y 354.811,Z 301.098,A -85,B 0,C 180,E1 -13355.699,E2 -13355.699} C_VEL
LIN {X 0,Y 354.762,Z 301.105,A -85,B 0,C 180,E1 -13359.413,E2 -13359.413} C_VEL
LIN {X 0,Y 354.775,Z 301.107,A -85,B 0,C 180,E1 -13362.866,E2 -13362.866} C_VEL
LIN {X 0,Y 354.757,Z 301.104,A -85,B 0,C 180,E1 -13366.103,E2 -13366.103} C_VEL
LIN {X 0,Y 354.758,Z 301.106,A -85,B 0,C 180,E1 -13369.176,E2 -13369.176} C_VEL
LIN {X 0,Y 354.795,Z 301.102,A -85,B 0,C 180,E1 -13372.405,E2 -13372.405} C_VEL
LIN {X 0,Y 354.807,Z 301.101,A -85,B 0,C 180,E1 -13374.941,E2 -13374.941} C_VEL
LIN {X 0,Y 354.79,Z 301.105,A -85,B 0,C 180,E1 -13378.406,E2 -13378.406} C_VEL
LIN {X 0,Y 354.794,Z 301.1,A -85,B 0,C 180,E1 -13381.615,E2 -13381.615} C_VEL
LIN {X 0,Y 354.907,Z 301.293,A -85,B 0,C 180,E1 -13385.272,E2 -13385.272} C_VEL
LIN {X 0,Y 356.329,Z 309.541,A -85,B 0,C 180,E1 -13387.992,E2 -13387.992} C_VEL
LIN {X 0,Y 356.467,Z 313.444,A -85,B 0,C 180,E1 -13389.214,E2 -13389.214} C_VEL
LIN {X 0,Y 355.683,Z 323.621,A -85,B 0,C 180,E1 -13392.24,E2 -13392.24} C_VEL
LIN {X 0,Y 356.236,Z 327.175,A -85,B 0,C 180,E1 -13392.411,E2 -13392.411} C_VEL
LIN {X 0,Y 359.791,Z 349.374,A -85,B 0,C 180,E1 -13393.045,E2 -13393.045} C_VEL
LIN {X 0,Y 359.209,Z 399.838,A -85,B 0,C 180,E1 -13394.079,E2 -13394.079} C_VEL
LIN {X 0,Y 358.801,Z 409.415,A -85,B 0,C 180,E1 -13394.413,E2 -13394.413} C_VEL
LIN {X 0,Y 358.328,Z 419.427,A -85,B 0,C 180,E1 -13394.938,E2 -13394.938} C_VEL
LIN {X 0,Y 357.544,Z 430.797,A -85,B 0,C 180,E1 -13395.777,E2 -13395.777} C_VEL
LIN {X 0,Y 356.834,Z 439.363,A -85,B 0,C 180,E1 -13396.62,E2 -13396.62} C_VEL
LIN {X 0,Y 356.16,Z 447.421,A -85,B 0,C 180,E1 -13397.609,E2 -13397.609} C_VEL
LIN {X 0,Y 355.516,Z 454.076,A -85,B 0,C 180,E1 -13398.599,E2 -13398.599} C_VEL
LIN {X 0,Y 354.921,Z 460.392,A -85,B 0,C 180,E1 -13399.734,E2 -13399.734} C_VEL
LIN {X 0,Y 354.378,Z 465.638,A -85,B 0,C 180,E1 -13400.871,E2 -13400.871} C_VEL
LIN {X 0,Y 354.009,Z 470.012,A -85,B 0,C 180,E1 -13402.012,E2 -13402.012} C_VEL
LIN {X 0,Y 353.632,Z 474.726,A -85,B 0,C 180,E1 -13403.558,E2 -13403.558} C_VEL
LIN {X 0,Y 353.488,Z 477.8,A -85,B 0,C 180,E1 -13404.867,E2 -13404.867} C_VEL
LIN {X 0,Y 353.259,Z 480.689,A -85,B 0,C 180,E1 -13406.578,E2 -13406.578} C_VEL
LIN {X 0,Y 353.177,Z 481.934,A -85,B 0,C 180,E1 -13407.719,E2 -13407.719} C_VEL
LIN {X 0,Y 353.155,Z 482.707,A -85,B 0,C 180,E1 -13408.86,E2 -13408.86} C_VEL
LIN {X 0,Y 353.141,Z 483,A -85,B 0,C 180,E1 -13410,E2 -13410} C_VEL
LIN {X 0,Y 353.155,Z 482.703,A -85,B 0,C 180,E1 -13411.14,E2 -13411.14} C_VEL
LIN {X 0,Y 353.177,Z 481.922,A -85,B 0,C 180,E1 -13412.281,E2 -13412.281} C_VEL
LIN {X 0,Y 353.258,Z 480.669,A -85,B 0,C 180,E1 -13413.422,E2 -13413.422} C_VEL
LIN {X 0,Y 353.482,Z 477.772,A -85,B 0,C 180,E1 -13415.133,E2 -13415.133} C_VEL
LIN {X 0,Y 353.669,Z 474.549,A -85,B 0,C 180,E1 -13416.494,E2 -13416.494} C_VEL
LIN {X 0,Y 354.094,Z 469.005,A -85,B 0,C 180,E1 -13418.273,E2 -13418.273} C_VEL
LIN {X 0,Y 354.625,Z 463.15,A -85,B 0,C 180,E1 -13419.698,E2 -13419.698} C_VEL
LIN {X 0,Y 355.351,Z 455.699,A -85,B 0,C 180,E1 -13421.118,E2 -13421.118} C_VEL
LIN {X 0,Y 356.081,Z 448.349,A -85,B 0,C 180,E1 -13422.249,E2 -13422.249} C_VEL
LIN {X 0,Y 356.711,Z 440.474,A -85,B 0,C 180,E1 -13423.24,E2 -13423.24} C_VEL
LIN {X 0,Y 357.414,Z 432.15,A -85,B 0,C 180,E1 -13424.083,E2 -13424.083} C_VEL
LIN {X 0,Y 358.178,Z 421.512,A -85,B 0,C 180,E1 -13424.923,E2 -13424.923} C_VEL
LIN {X 0,Y 358.756,Z 409.918,A -85,B 0,C 180,E1 -13425.553,E2 -13425.553} C_VEL
LIN {X 0,Y 359.142,Z 400.192,A -85,B 0,C 180,E1 -13425.9,E2 -13425.9} C_VEL
LIN {X 0,Y 359.73,Z 348.371,A -85,B 0,C 180,E1 -13426.964,E2 -13426.964} C_VEL
LIN {X 0,Y 355.709,Z 324.257,A -85,B 0,C 180,E1 -13427.68,E2 -13427.68} C_VEL
LIN {X 0,Y 355.695,Z 323.239,A -85,B 0,C 180,E1 -13427.833,E2 -13427.833} C_VEL
LIN {X 0,Y 356.457,Z 313.391,A -85,B 0,C 180,E1 -13430.786,E2 -13430.786} C_VEL
LIN {X 0,Y 356.314,Z 309.443,A -85,B 0,C 180,E1 -13432.023,E2 -13432.023} C_VEL
LIN {X 0,Y 354.87,Z 301.183,A -85,B 0,C 180,E1 -13434.809,E2 -13434.809} C_VEL
LIN {X 0,Y 354.796,Z 301.099,A -85,B 0,C 180,E1 -13438.385,E2 -13438.385} C_VEL
LIN {X 0,Y 354.783,Z 301.101,A -85,B 0,C 180,E1 -13442.333,E2 -13442.333} C_VEL
LIN {X 0,Y 354.817,Z 301.099,A -85,B 0,C 180,E1 -13445.698,E2 -13445.698} C_VEL
LIN {X 0,Y 354.764,Z 301.107,A -85,B 0,C 180,E1 -13449.412,E2 -13449.412} C_VEL
LIN {X 0,Y 354.776,Z 301.104,A -85,B 0,C 180,E1 -13452.865,E2 -13452.865} C_VEL
LIN {X 0,Y 354.756,Z 301.104,A -85,B 0,C 180,E1 -13456.102,E2 -13456.102} C_VEL
LIN {X 0,Y 354.757,Z 301.107,A -85,B 0,C 180,E1 -13459.175,E2 -13459.175} C_VEL
LIN {X 0,Y 354.793,Z 301.1,A -85,B 0,C 180,E1 -13462.404,E2 -13462.404} C_VEL
LIN {X 0,Y 354.801,Z 301.104,A -85,B 0,C 180,E1 -13464.94,E2 -13464.94} C_VEL
LIN {X 0,Y 354.786,Z 301.103,A -85,B 0,C 180,E1 -13468.405,E2 -13468.405} C_VEL
LIN {X 0,Y 354.789,Z 301.1,A -85,B 0,C 180,E1 -13471.614,E2 -13471.614} C_VEL
LIN {X 0,Y 354.796,Z 301.099,A -85,B 0,C 180,E1 -13475.419,E2 -13475.419} C_VEL
LIN {X 0,Y 354.812,Z 301.098,A -85,B 0,C 180,E1 -13479.112,E2 -13479.112} C_VEL
LIN {X 0,Y 354.842,Z 301.097,A -85,B 0,C 180,E1 -13482.717,E2 -13482.717} C_VEL
LIN {X 0,Y 354.931,Z 301.087,A -85,B 0,C 180,E1 -13486.254,E2 -13486.254} C_VEL
LIN {X 0,Y 354.946,Z 301.082,A -85,B 0,C 180,E1 -13489.735,E2 -13489.735} C_VEL
LIN {X 0,Y 355.078,Z 301.064,A -85,B 0,C 180,E1 -13493.18,E2 -13493.18} C_VEL
LIN {X 0,Y 355.216,Z 301.049,A -85,B 0,C 180,E1 -13497.732,E2 -13497.732} C_VEL
LIN {X 0,Y 355.135,Z 301.057,A -85,B 0,C 180,E1 -13501.134,E2 -13501.134} C_VEL
LIN {X 0,Y 355.21,Z 301.05,A -85,B 0,C 180,E1 -13502.268,E2 -13502.268} C_VEL
LIN {X 0,Y 355.078,Z 301.064,A -85,B 0,C 180,E1 -13506.821,E2 -13506.821} C_VEL
LIN {X 0,Y 354.941,Z 301.083,A -85,B 0,C 180,E1 -13510.265,E2 -13510.265} C_VEL
LIN {X 0,Y 354.915,Z 301.087,A -85,B 0,C 180,E1 -13514.006,E2 -13514.006} C_VEL
LIN {X 0,Y 354.836,Z 301.096,A -85,B 0,C 180,E1 -13518.069,E2 -13518.069} C_VEL
LIN {X 0,Y 354.798,Z 301.099,A -85,B 0,C 180,E1 -13522.109,E2 -13522.109} C_VEL
LIN {X 0,Y 354.788,Z 301.102,A -85,B 0,C 180,E1 -13525.836,E2 -13525.836} C_VEL
LIN {X 0,Y 354.786,Z 301.102,A -85,B 0,C 180,E1 -13529.685,E2 -13529.685} C_VEL
LIN {X 0,Y 354.78,Z 301.101,A -85,B 0,C 180,E1 -13532.334,E2 -13532.334} C_VEL
LIN {X 0,Y 354.812,Z 301.098,A -85,B 0,C 180,E1 -13535.699,E2 -13535.699} C_VEL
LIN {X 0,Y 354.763,Z 301.105,A -85,B 0,C 180,E1 -13539.413,E2 -13539.413} C_VEL
LIN {X 0,Y 354.776,Z 301.106,A -85,B 0,C 180,E1 -13542.867,E2 -13542.867} C_VEL
LIN {X 0,Y 354.758,Z 301.104,A -85,B 0,C 180,E1 -13546.104,E2 -13546.104} C_VEL
LIN {X 0,Y 354.759,Z 301.106,A -85,B 0,C 180,E1 -13549.176,E2 -13549.176} C_VEL
LIN {X 0,Y 354.797,Z 301.102,A -85,B 0,C 180,E1 -13552.405,E2 -13552.405} C_VEL
LIN {X 0,Y 354.808,Z 301.101,A -85,B 0,C 180,E1 -13554.941,E2 -13554.941} C_VEL
LIN {X 0,Y 354.791,Z 301.104,A -85,B 0,C 180,E1 -13558.406,E2 -13558.406} C_VEL
LIN {X 0,Y 354.787,Z 301.101,A -85,B 0,C 180,E1 -13561.614,E2 -13561.614} C_VEL
LIN {X 0,Y 354.923,Z 301.321,A -85,B 0,C 180,E1 -13565.351,E2 -13565.351} C_VEL
LIN {X 0,Y 356.322,Z 309.343,A -85,B 0,C 180,E1 -13567.992,E2 -13567.992} C_VEL
LIN {X 0,Y 356.314,Z 315.198,A -85,B 0,C 180,E1 -13569.808,E2 -13569.808} C_VEL
LIN {X 0,Y 355.68,Z 323.702,A -85,B 0,C 180,E1 -13572.309,E2 -13572.309} C_VEL
LIN {X 0,Y 356.314,Z 327.802,A -85,B 0,C 180,E1 -13572.488,E2 -13572.488} C_VEL
LIN {X 0,Y 359.786,Z 349.567,A -85,B 0,C 180,E1 -13573.108,E2 -13573.108} C_VEL
LIN {X 0,Y 359.137,Z 399.887,A -85,B 0,C 180,E1 -13574.136,E2 -13574.136} C_VEL
LIN {X 0,Y 358.833,Z 408.89,A -85,B 0,C 180,E1 -13574.45,E2 -13574.45} C_VEL
LIN {X 0,Y 358.341,Z 418.442,A -85,B 0,C 180,E1 -13574.938,E2 -13574.938} C_VEL
LIN {X 0,Y 357.72,Z 428.465,A -85,B 0,C 180,E1 -13575.639,E2 -13575.639} C_VEL
LIN {X 0,Y 356.897,Z 438.862,A -85,B 0,C 180,E1 -13576.622,E2 -13576.622} C_VEL
LIN {X 0,Y 356.185,Z 447.01,A -85,B 0,C 180,E1 -13577.61,E2 -13577.61} C_VEL
LIN {X 0,Y 355.546,Z 453.733,A -85,B 0,C 180,E1 -13578.6,E2 -13578.6} C_VEL
LIN {X 0,Y 354.924,Z 460.099,A -85,B 0,C 180,E1 -13579.735,E2 -13579.735} C_VEL
LIN {X 0,Y 354.435,Z 465.393,A -85,B 0,C 180,E1 -13580.873,E2 -13580.873} C_VEL
LIN {X 0,Y 354.053,Z 469.813,A -85,B 0,C 180,E1 -13582.013,E2 -13582.013} C_VEL
LIN {X 0,Y 353.672,Z 474.423,A -85,B 0,C 180,E1 -13583.503,E2 -13583.503} C_VEL
LIN {X 0,Y 353.49,Z 477.682,A -85,B 0,C 180,E1 -13584.867,E2 -13584.867} C_VEL
LIN {X 0,Y 353.261,Z 480.606,A -85,B 0,C 180,E1 -13586.578,E2 -13586.578} C_VEL
LIN {X 0,Y 353.178,Z 481.884,A -85,B 0,C 180,E1 -13587.719,E2 -13587.719} C_VEL
LIN {X 0,Y 353.156,Z 482.691,A -85,B 0,C 180,E1 -13588.86,E2 -13588.86} C_VEL
LIN {X 0,Y 353.142,Z 482.998,A -85,B 0,C 180,E1 -13590,E2 -13590} C_VEL
LIN {X 0,Y 353.152,Z 482.72,A -85,B 0,C 180,E1 -13591.14,E2 -13591.14} C_VEL
LIN {X 0,Y 353.164,Z 481.972,A -85,B 0,C 180,E1 -13592.281,E2 -13592.281} C_VEL
LIN {X 0,Y 353.255,Z 480.753,A -85,B 0,C 180,E1 -13593.422,E2 -13593.422} C_VEL
LIN {X 0,Y 353.476,Z 477.891,A -85,B 0,C 180,E1 -13595.133,E2 -13595.133} C_VEL
LIN {X 0,Y 353.602,Z 474.966,A -85,B 0,C 180,E1 -13596.397,E2 -13596.397} C_VEL
LIN {X 0,Y 354.002,Z 470.162,A -85,B 0,C 180,E1 -13597.988,E2 -13597.988} C_VEL
LIN {X 0,Y 354.483,Z 464.649,A -85,B 0,C 180,E1 -13599.414,E2 -13599.414} C_VEL
LIN {X 0,Y 355.181,Z 457.727,A -85,B 0,C 180,E1 -13600.835,E2 -13600.835} C_VEL
LIN {X 0,Y 355.948,Z 449.78,A -85,B 0,C 180,E1 -13602.109,E2 -13602.109} C_VEL
LIN {X 0,Y 356.584,Z 442.203,A -85,B 0,C 180,E1 -13603.1,E2 -13603.1} C_VEL
LIN {X 0,Y 357.358,Z 434.263,A -85,B 0,C 180,E1 -13603.94,E2 -13603.94} C_VEL
LIN {X 0,Y 357.929,Z 426.064,A -85,B 0,C 180,E1 -13604.643,E2 -13604.643} C_VEL
LIN {X 0,Y 358.43,Z 417.756,A -85,B 0,C 180,E1 -13605.203,E2 -13605.203} C_VEL
LIN {X 0,Y 358.83,Z 408.779,A -85,B 0,C 180,E1 -13605.659,E2 -13605.659} C_VEL
LIN {X 0,Y 359.191,Z 399.415,A -85,B 0,C 180,E1 -13605.979,E2 -13605.979} C_VEL
LIN {X 0,Y 359.685,Z 348.349,A -85,B 0,C 180,E1 -13607.026,E2 -13607.026} C_VEL
LIN {X 0,Y 355.845,Z 324.931,A -85,B 0,C 180,E1 -13607.712,E2 -13607.712} C_VEL
LIN {X 0,Y 355.326,Z 323.294,A -85,B 0,C 180,E1 -13607.916,E2 -13607.916} C_VEL
LIN {X 0,Y 352.115,Z 318.438,A -85,B 0,C 180,E1 -13609.54,E2 -13609.54} C_VEL
LIN {X 0,Y 350.26,Z 314.854,A -85,B 0,C 180,E1 -13610.87,E2 -13610.87} C_VEL
LIN {X 0,Y 349.309,Z 310.597,A -85,B 0,C 180,E1 -13612.182,E2 -13612.182} C_VEL
LIN {X 0,Y 347.834,Z 302.071,A -85,B 0,C 180,E1 -13615.106,E2 -13615.106} C_VEL
LIN {X 0,Y 347.743,Z 301.979,A -85,B 0,C 180,E1 -13619.015,E2 -13619.015} C_VEL
LIN {X 0,Y 347.737,Z 301.981,A -85,B 0,C 180,E1 -13621.913,E2 -13621.913} C_VEL
LIN {X 0,Y 347.785,Z 301.974,A -85,B 0,C 180,E1 -13625.875,E2 -13625.875} C_VEL
LIN {X 0,Y 347.728,Z 301.981,A -85,B 0,C 180,E1 -13628.795,E2 -13628.795} C_VEL
LIN {X 0,Y 347.736,Z 301.978,A -85,B 0,C 180,E1 -13631.831,E2 -13631.831} C_VEL
LIN {X 0,Y 347.696,Z 301.988,A -85,B 0,C 180,E1 -13635.027,E2 -13635.027} C_VEL
LIN {X 0,Y 347.735,Z 301.979,A -85,B 0,C 180,E1 -13638.399,E2 -13638.399} C_VEL
LIN {X 0,Y 347.757,Z 301.973,A -85,B 0,C 180,E1 -13642.013,E2 -13642.013} C_VEL
LIN {X 0,Y 347.737,Z 301.979,A -85,B 0,C 180,E1 -13645.535,E2 -13645.535} C_VEL
LIN {X 0,Y 347.738,Z 301.98,A -85,B 0,C 180,E1 -13648.3,E2 -13648.3} C_VEL
LIN {X 0,Y 347.738,Z 301.982,A -85,B 0,C 180,E1 -13650.984,E2 -13650.984} C_VEL
LIN {X 0,Y 347.727,Z 301.98,A -85,B 0,C 180,E1 -13653.599,E2 -13653.599} C_VEL
LIN {X 0,Y 347.741,Z 301.98,A -85,B 0,C 180,E1 -13656.158,E2 -13656.158} C_VEL
LIN {X 0,Y 347.763,Z 301.976,A -85,B 0,C 180,E1 -13659.906,E2 -13659.906} C_VEL
LIN {X 0,Y 347.788,Z 301.972,A -85,B 0,C 180,E1 -13663.566,E2 -13663.566} C_VEL
LIN {X 0,Y 347.878,Z 301.96,A -85,B 0,C 180,E1 -13667.16,E2 -13667.16} C_VEL
LIN {X 0,Y 347.927,Z 301.957,A -85,B 0,C 180,E1 -13670.7,E2 -13670.7} C_VEL
LIN {X 0,Y 348.03,Z 301.946,A -85,B 0,C 180,E1 -13674.205,E2 -13674.205} C_VEL
LIN {X 0,Y 348.178,Z 301.925,A -85,B 0,C 180,E1 -13677.686,E2 -13677.686} C_VEL
LIN {X 0,Y 348.106,Z 301.933,A -85,B 0,C 180,E1 -13681.157,E2 -13681.157} C_VEL
LIN {X 0,Y 348.171,Z 301.926,A -85,B 0,C 180,E1 -13682.314,E2 -13682.314} C_VEL
LIN {X 0,Y 348.045,Z 301.94,A -85,B 0,C 180,E1 -13686.959,E2 -13686.959} C_VEL
LIN {X 0,Y 347.881,Z 301.961,A -85,B 0,C 180,E1 -13690.476,E2 -13690.476} C_VEL
LIN {X 0,Y 347.872,Z 301.962,A -85,B 0,C 180,E1 -13694.137,E2 -13694.137} C_VEL
LIN {X 0,Y 347.786,Z 301.973,A -85,B 0,C 180,E1 -13698.242,E2 -13698.242} C_VEL
LIN {X 0,Y 347.755,Z 301.979,A -85,B 0,C 180,E1 -13701.624,E2 -13701.624} C_VEL
LIN {X 0,Y 347.729,Z 301.983,A -85,B 0,C 180,E1 -13705.115,E2 -13705.115} C_VEL
LIN {X 0,Y 347.721,Z 301.983,A -85,B 0,C 180,E1 -13707.701,E2 -13707.701} C_VEL
LIN {X 0,Y 347.731,Z 301.978,A -85,B 0,C 180,E1 -13710.35,E2 -13710.35} C_VEL
LIN {X 0,Y 347.742,Z 301.978,A -85,B 0,C 180,E1 -13714.044,E2 -13714.044} C_VEL
LIN {X 0,Y 347.748,Z 301.978,A -85,B 0,C 180,E1 -13717.322,E2 -13717.322} C_VEL
LIN {X 0,Y 347.69,Z 301.982,A -85,B 0,C 180,E1 -13720.303,E2 -13720.303} C_VEL
LIN {X 0,Y 347.715,Z 301.983,A -85,B 0,C 180,E1 -13723.409,E2 -13723.409} C_VEL
LIN {X 0,Y 347.717,Z 301.985,A -85,B 0,C 180,E1 -13726.688,E2 -13726.688} C_VEL
LIN {X 0,Y 347.696,Z 301.983,A -85,B 0,C 180,E1 -13730.183,E2 -13730.183} C_VEL
LIN {X 0,Y 347.752,Z 301.983,A -85,B 0,C 180,E1 -13732.679,E2 -13732.679} C_VEL
LIN {X 0,Y 347.745,Z 301.978,A -85,B 0,C 180,E1 -13735.957,E2 -13735.957} C_VEL
LIN {X 0,Y 347.735,Z 301.979,A -85,B 0,C 180,E1 -13739.652,E2 -13739.652} C_VEL
LIN {X 0,Y 347.738,Z 301.974,A -85,B 0,C 180,E1 -13743.601,E2 -13743.601} C_VEL
LIN {X 0,Y 347.844,Z 302.216,A -85,B 0,C 180,E1 -13745.043,E2 -13745.043} C_VEL
LIN {X 0,Y 349.284,Z 310.264,A -85,B 0,C 180,E1 -13747.755,E2 -13747.755} C_VEL
LIN {X 0,Y 349.396,Z 315.398,A -85,B 0,C 180,E1 -13749.39,E2 -13749.39} C_VEL
LIN {X 0,Y 348.757,Z 323.817,A -85,B 0,C 180,E1 -13751.902,E2 -13751.902} C_VEL
LIN {X 0,Y 350.161,Z 331.772,A -85,B 0,C 180,E1 -13752.192,E2 -13752.192} C_VEL
LIN {X 0,Y 353.009,Z 349.887,A -85,B 0,C 180,E1 -13752.719,E2 -13752.719} C_VEL
LIN {X 0,Y 352.384,Z 399.897,A -85,B 0,C 180,E1 -13753.763,E2 -13753.763} C_VEL
LIN {X 0,Y 351.978,Z 409.424,A -85,B 0,C 180,E1 -13754.102,E2 -13754.102} C_VEL
LIN {X 0,Y 351.478,Z 419.434,A -85,B 0,C 180,E1 -13754.637,E2 -13754.637} C_VEL
LIN {X 0,Y 350.661,Z 430.801,A -85,B 0,C 180,E1 -13755.492,E2 -13755.492} C_VEL
LIN {X 0,Y 349.94,Z 439.367,A -85,B 0,C 180,E1 -13756.351,E2 -13756.351} C_VEL
LIN {X 0,Y 349.222,Z 447.424,A -85,B 0,C 180,E1 -13757.358,E2 -13757.358} C_VEL
LIN {X 0,Y 348.557,Z 454.078,A -85,B 0,C 180,E1 -13758.368,E2 -13758.368} C_VEL
LIN {X 0,Y 347.938,Z 460.394,A -85,B 0,C 180,E1 -13759.526,E2 -13759.526} C_VEL
LIN {X 0,Y 347.361,Z 465.64,A -85,B 0,C 180,E1 -13760.685,E2 -13760.685} C_VEL
LIN {X 0,Y 346.98,Z 470.013,A -85,B 0,C 180,E1 -13761.849,E2 -13761.849} C_VEL
LIN {X 0,Y 346.523,Z 475.209,A -85,B 0,C 180,E1 -13763.611,E2 -13763.611} C_VEL
LIN {X 0,Y 346.334,Z 478.952,A -85,B 0,C 180,E1 -13765.344,E2 -13765.344} C_VEL
LIN {X 0,Y 346.186,Z 480.69,A -85,B 0,C 180,E1 -13766.508,E2 -13766.508} C_VEL
LIN {X 0,Y 346.089,Z 481.934,A -85,B 0,C 180,E1 -13767.672,E2 -13767.672} C_VEL
LIN {X 0,Y 346.058,Z 482.708,A -85,B 0,C 180,E1 -13768.836,E2 -13768.836} C_VEL
LIN {X 0,Y 346.043,Z 483,A -85,B 0,C 180,E1 -13770,E2 -13770} C_VEL
LIN {X 0,Y 346.058,Z 482.703,A -85,B 0,C 180,E1 -13771.164,E2 -13771.164} C_VEL
LIN {X 0,Y 346.089,Z 481.921,A -85,B 0,C 180,E1 -13772.328,E2 -13772.328} C_VEL
LIN {X 0,Y 346.186,Z 480.669,A -85,B 0,C 180,E1 -13773.492,E2 -13773.492} C_VEL
LIN {X 0,Y 346.388,Z 477.772,A -85,B 0,C 180,E1 -13775.238,E2 -13775.238} C_VEL
LIN {X 0,Y 346.555,Z 475.049,A -85,B 0,C 180,E1 -13776.435,E2 -13776.435} C_VEL
LIN {X 0,Y 346.972,Z 469.962,A -85,B 0,C 180,E1 -13778.151,E2 -13778.151} C_VEL
LIN {X 0,Y 347.607,Z 463.148,A -85,B 0,C 180,E1 -13779.895,E2 -13779.895} C_VEL
LIN {X 0,Y 348.373,Z 455.697,A -85,B 0,C 180,E1 -13781.343,E2 -13781.343} C_VEL
LIN {X 0,Y 349.141,Z 448.346,A -85,B 0,C 180,E1 -13782.497,E2 -13782.497} C_VEL
LIN {X 0,Y 349.799,Z 440.471,A -85,B 0,C 180,E1 -13783.507,E2 -13783.507} C_VEL
LIN {X 0,Y 350.55,Z 432.146,A -85,B 0,C 180,E1 -13784.365,E2 -13784.365} C_VEL
LIN {X 0,Y 351.324,Z 421.506,A -85,B 0,C 180,E1 -13785.221,E2 -13785.221} C_VEL
LIN {X 0,Y 351.932,Z 409.909,A -85,B 0,C 180,E1 -13785.862,E2 -13785.862} C_VEL
LIN {X 0,Y 352.328,Z 400.177,A -85,B 0,C 180,E1 -13786.216,E2 -13786.216} C_VEL
LIN {X 0,Y 352.969,Z 349.154,A -85,B 0,C 180,E1 -13787.282,E2 -13787.282} C_VEL
LIN {X 0,Y 348.762,Z 324.136,A -85,B 0,C 180,E1 -13788.05,E2 -13788.05} C_VEL
LIN {X 0,Y 348.745,Z 323.359,A -85,B 0,C 180,E1 -13788.169,E2 -13788.169} C_VEL
LIN {X 0,Y 349.49,Z 313.39,A -85,B 0,C 180,E1 -13791.221,E2 -13791.221} C_VEL
LIN {X 0,Y 348.834,Z 307.533,A -85,B 0,C 180,E1 -13793.133,E2 -13793.133} C_VEL
LIN {X 0,Y 347.834,Z 302.074,A -85,B 0,C 180,E1 -13795.032,E2 -13795.032} C_VEL
LIN {X 0,Y 347.742,Z 301.98,A -85,B 0,C 180,E1 -13799.015,E2 -13799.015} C_VEL
LIN {X 0,Y 347.735,Z 301.981,A -85,B 0,C 180,E1 -13801.913,E2 -13801.913} C_VEL
LIN {X 0,Y 347.783,Z 301.974,A -85,B 0,C 180,E1 -13805.875,E2 -13805.875} C_VEL
LIN {X 0,Y 347.726,Z 301.982,A -85,B 0,C 180,E1 -13808.795,E2 -13808.795} C_VEL
LIN {X 0,Y 347.735,Z 301.978,A -85,B 0,C 180,E1 -13811.831,E2 -13811.831} C_VEL
LIN {X 0,Y 347.695,Z 301.989,A -85,B 0,C 180,E1 -13815.027,E2 -13815.027} C_VEL
LIN {X 0,Y 347.732,Z 301.979,A -85,B 0,C 180,E1 -13818.399,E2 -13818.399} C_VEL
LIN {X 0,Y 347.756,Z 301.973,A -85,B 0,C 180,E1 -13822.013,E2 -13822.013} C_VEL
LIN {X 0,Y 347.736,Z 301.979,A -85,B 0,C 180,E1 -13825.535,E2 -13825.535} C_VEL
LIN {X 0,Y 347.737,Z 301.98,A -85,B 0,C 180,E1 -13828.3,E2 -13828.3} C_VEL
LIN {X 0,Y 347.737,Z 301.982,A -85,B 0,C 180,E1 -13830.984,E2 -13830.984} C_VEL
LIN {X 0,Y 347.726,Z 301.98,A -85,B 0,C 180,E1 -13833.599,E2 -13833.599} C_VEL
LIN {X 0,Y 347.74,Z 301.98,A -85,B 0,C 180,E1 -13836.159,E2 -13836.159} C_VEL
LIN {X 0,Y 347.762,Z 301.976,A -85,B 0,C 180,E1 -13839.906,E2 -13839.906} C_VEL
LIN {X 0,Y 347.788,Z 301.972,A -85,B 0,C 180,E1 -13843.566,E2 -13843.566} C_VEL
LIN {X 0,Y 347.878,Z 301.96,A -85,B 0,C 180,E1 -13847.16,E2 -13847.16} C_VEL
LIN {X 0,Y 347.926,Z 301.957,A -85,B 0,C 180,E1 -13850.7,E2 -13850.7} C_VEL
LIN {X 0,Y 348.029,Z 301.946,A -85,B 0,C 180,E1 -13854.205,E2 -13854.205} C_VEL
LIN {X 0,Y 348.177,Z 301.925,A -85,B 0,C 180,E1 -13857.686,E2 -13857.686} C_VEL
LIN {X 0,Y 348.106,Z 301.933,A -85,B 0,C 180,E1 -13861.157,E2 -13861.157} C_VEL
LIN {X 0,Y 348.171,Z 301.926,A -85,B 0,C 180,E1 -13862.314,E2 -13862.314} C_VEL
LIN {X 0,Y 348.045,Z 301.94,A -85,B 0,C 180,E1 -13866.959,E2 -13866.959} C_VEL
LIN {X 0,Y 347.881,Z 301.961,A -85,B 0,C 180,E1 -13870.476,E2 -13870.476} C_VEL
LIN {X 0,Y 347.872,Z 301.962,A -85,B 0,C 180,E1 -13874.138,E2 -13874.138} C_VEL
LIN {X 0,Y 347.787,Z 301.973,A -85,B 0,C 180,E1 -13878.242,E2 -13878.242} C_VEL
LIN {X 0,Y 347.756,Z 301.979,A -85,B 0,C 180,E1 -13881.625,E2 -13881.625} C_VEL
LIN {X 0,Y 347.727,Z 301.983,A -85,B 0,C 180,E1 -13885.115,E2 -13885.115} C_VEL
LIN {X 0,Y 347.718,Z 301.983,A -85,B 0,C 180,E1 -13887.702,E2 -13887.702} C_VEL
LIN {X 0,Y 347.729,Z 301.979,A -85,B 0,C 180,E1 -13890.35,E2 -13890.35} C_VEL
LIN {X 0,Y 347.742,Z 301.978,A -85,B 0,C 180,E1 -13894.044,E2 -13894.044} C_VEL
LIN {X 0,Y 347.749,Z 301.978,A -85,B 0,C 180,E1 -13897.323,E2 -13897.323} C_VEL
LIN {X 0,Y 347.691,Z 301.982,A -85,B 0,C 180,E1 -13900.303,E2 -13900.303} C_VEL
LIN {X 0,Y 347.716,Z 301.983,A -85,B 0,C 180,E1 -13903.409,E2 -13903.409} C_VEL
LIN {X 0,Y 347.718,Z 301.985,A -85,B 0,C 180,E1 -13906.688,E2 -13906.688} C_VEL
LIN {X 0,Y 347.697,Z 301.983,A -85,B 0,C 180,E1 -13910.183,E2 -13910.183} C_VEL
LIN {X 0,Y 347.753,Z 301.982,A -85,B 0,C 180,E1 -13912.679,E2 -13912.679} C_VEL
LIN {X 0,Y 347.746,Z 301.977,A -85,B 0,C 180,E1 -13915.957,E2 -13915.957} C_VEL
LIN {X 0,Y 347.734,Z 301.979,A -85,B 0,C 180,E1 -13919.651,E2 -13919.651} C_VEL
LIN {X 0,Y 347.739,Z 301.975,A -85,B 0,C 180,E1 -13923.601,E2 -13923.601} C_VEL
LIN {X 0,Y 347.858,Z 302.241,A -85,B 0,C 180,E1 -13925.12,E2 -13925.12} C_VEL
LIN {X 0,Y 349.276,Z 310.08,A -85,B 0,C 180,E1 -13927.758,E2 -13927.758} C_VEL
LIN {X 0,Y 349.39,Z 315.2,A -85,B 0,C 180,E1 -13929.39,E2 -13929.39} C_VEL
LIN {X 0,Y 348.732,Z 323.721,A -85,B 0,C 180,E1 -13931.947,E2 -13931.947} C_VEL
LIN {X 0,Y 349.441,Z 328.021,A -85,B 0,C 180,E1 -13932.136,E2 -13932.136} C_VEL
LIN {X 0,Y 353.009,Z 350.125,A -85,B 0,C 180,E1 -13932.785,E2 -13932.785} C_VEL
LIN {X 0,Y 352.331,Z 399.905,A -85,B 0,C 180,E1 -13933.822,E2 -13933.822} C_VEL
LIN {X 0,Y 351.999,Z 408.902,A -85,B 0,C 180,E1 -13934.141,E2 -13934.141} C_VEL
LIN {X 0,Y 351.494,Z 418.45,A -85,B 0,C 180,E1 -13934.638,E2 -13934.638} C_VEL
LIN {X 0,Y 350.854,Z 428.472,A -85,B 0,C 180,E1 -13935.352,E2 -13935.352} C_VEL
LIN {X 0,Y 350.009,Z 438.867,A -85,B 0,C 180,E1 -13936.354,E2 -13936.354} C_VEL
LIN {X 0,Y 349.227,Z 447.014,A -85,B 0,C 180,E1 -13937.359,E2 -13937.359} C_VEL
LIN {X 0,Y 348.593,Z 453.736,A -85,B 0,C 180,E1 -13938.369,E2 -13938.369} C_VEL
LIN {X 0,Y 347.928,Z 460.102,A -85,B 0,C 180,E1 -13939.526,E2 -13939.526} C_VEL
LIN {X 0,Y 347.295,Z 466.568,A -85,B 0,C 180,E1 -13940.977,E2 -13940.977} C_VEL
LIN {X 0,Y 346.872,Z 471.728,A -85,B 0,C 180,E1 -13942.433,E2 -13942.433} C_VEL
LIN {X 0,Y 346.439,Z 476.504,A -85,B 0,C 180,E1 -13944.179,E2 -13944.179} C_VEL
LIN {X 0,Y 346.351,Z 478.833,A -85,B 0,C 180,E1 -13945.345,E2 -13945.345} C_VEL
LIN {X 0,Y 346.19,Z 480.606,A -85,B 0,C 180,E1 -13946.508,E2 -13946.508} C_VEL
LIN {X 0,Y 346.091,Z 481.884,A -85,B 0,C 180,E1 -13947.672,E2 -13947.672} C_VEL
LIN {X 0,Y 346.059,Z 482.691,A -85,B 0,C 180,E1 -13948.836,E2 -13948.836} C_VEL
LIN {X 0,Y 346.044,Z 482.998,A -85,B 0,C 180,E1 -13950,E2 -13950} C_VEL
LIN {X 0,Y 346.055,Z 482.72,A -85,B 0,C 180,E1 -13951.164,E2 -13951.164} C_VEL
LIN {X 0,Y 346.077,Z 481.971,A -85,B 0,C 180,E1 -13952.328,E2 -13952.328} C_VEL
LIN {X 0,Y 346.182,Z 480.752,A -85,B 0,C 180,E1 -13953.492,E2 -13953.492} C_VEL
LIN {X 0,Y 346.382,Z 477.89,A -85,B 0,C 180,E1 -13955.238,E2 -13955.238} C_VEL
LIN {X 0,Y 346.519,Z 475.349,A -85,B 0,C 180,E1 -13956.38,E2 -13956.38} C_VEL
LIN {X 0,Y 346.973,Z 470.16,A -85,B 0,C 180,E1 -13958.151,E2 -13958.151} C_VEL
LIN {X 0,Y 347.48,Z 464.647,A -85,B 0,C 180,E1 -13959.605,E2 -13959.605} C_VEL
LIN {X 0,Y 348.212,Z 457.724,A -85,B 0,C 180,E1 -13961.054,E2 -13961.054} C_VEL
LIN {X 0,Y 349.013,Z 449.776,A -85,B 0,C 180,E1 -13962.354,E2 -13962.354} C_VEL
LIN {X 0,Y 349.689,Z 442.198,A -85,B 0,C 180,E1 -13963.363,E2 -13963.363} C_VEL
LIN {X 0,Y 350.472,Z 434.258,A -85,B 0,C 180,E1 -13964.22,E2 -13964.22} C_VEL
LIN {X 0,Y 351.081,Z 426.057,A -85,B 0,C 180,E1 -13964.935,E2 -13964.935} C_VEL
LIN {X 0,Y 351.603,Z 417.748,A -85,B 0,C 180,E1 -13965.506,E2 -13965.506} C_VEL
LIN {X 0,Y 352.01,Z 408.768,A -85,B 0,C 180,E1 -13965.97,E2 -13965.97} C_VEL
LIN {X 0,Y 352.379,Z 399.547,A -85,B 0,C 180,E1 -13966.292,E2 -13966.292} C_VEL
LIN {X 0,Y 352.942,Z 349.404,A -85,B 0,C 180,E1 -13967.339,E2 -13967.339} C_VEL
LIN {X 0,Y 348.835,Z 324.525,A -85,B 0,C 180,E1 -13968.092,E2 -13968.092} C_VEL
LIN {X 0,Y 348.738,Z 323.402,A -85,B 0,C 180,E1 -13968.22,E2 -13968.22} C_VEL
LIN {X 0,Y 349.476,Z 313.588,A -85,B 0,C 180,E1 -13971.221,E2 -13971.221} C_VEL
LIN {X 0,Y 349.309,Z 310.597,A -85,B 0,C 180,E1 -13972.182,E2 -13972.182} C_VEL
LIN {X 0,Y 348.444,Z 308.984,A -85,B 0,C 180,E1 -13972.757,E2 -13972.757} C_VEL
LIN {X 0,Y 345.231,Z 306.876,A -85,B 0,C 180,E1 -13973.666,E2 -13973.666} C_VEL
LIN {X 0,Y 341.878,Z 304.821,A -85,B 0,C 180,E1 -13974.593,E2 -13974.593} C_VEL
LIN {X 0,Y 340.829,Z 303.276,A -85,B 0,C 180,E1 -13975.191,E2 -13975.191} C_VEL
LIN {X 0,Y 340.75,Z 302.844,A -85,B 0,C 180,E1 -13975.666,E2 -13975.666} C_VEL
LIN {X 0,Y 340.72,Z 302.854,A -85,B 0,C 180,E1 -13979.965,E2 -13979.965} C_VEL
LIN {X 0,Y 340.69,Z 302.857,A -85,B 0,C 180,E1 -13983.846,E2 -13983.846} C_VEL
LIN {X 0,Y 340.699,Z 302.856,A -85,B 0,C 180,E1 -13986.741,E2 -13986.741} C_VEL
LIN {X 0,Y 340.647,Z 302.86,A -85,B 0,C 180,E1 -13990.238,E2 -13990.238} C_VEL
LIN {X 0,Y 340.668,Z 302.859,A -85,B 0,C 180,E1 -13992.904,E2 -13992.904} C_VEL
LIN {X 0,Y 340.668,Z 302.864,A -85,B 0,C 180,E1 -13997.094,E2 -13997.094} C_VEL
LIN {X 0,Y 340.65,Z 302.857,A -85,B 0,C 180,E1 -14000.24,E2 -14000.24} C_VEL
LIN {X 0,Y 340.701,Z 302.854,A -85,B 0,C 180,E1 -14003.56,E2 -14003.56} C_VEL
LIN {X 0,Y 340.687,Z 302.857,A -85,B 0,C 180,E1 -14006.153,E2 -14006.153} C_VEL
LIN {X 0,Y 340.715,Z 302.852,A -85,B 0,C 180,E1 -14010.034,E2 -14010.034} C_VEL
LIN {X 0,Y 340.703,Z 302.858,A -85,B 0,C 180,E1 -14013.011,E2 -14013.011} C_VEL
LIN {X 0,Y 340.693,Z 302.857,A -85,B 0,C 180,E1 -14016.924,E2 -14016.924} C_VEL
LIN {X 0,Y 340.696,Z 302.86,A -85,B 0,C 180,E1 -14020.728,E2 -14020.728} C_VEL
LIN {X 0,Y 340.784,Z 302.848,A -85,B 0,C 180,E1 -14024.449,E2 -14024.449} C_VEL
LIN {X 0,Y 340.84,Z 302.84,A -85,B 0,C 180,E1 -14028.1,E2 -14028.1} C_VEL
LIN {X 0,Y 340.972,Z 302.823,A -85,B 0,C 180,E1 -14031.704,E2 -14031.704} C_VEL
LIN {X 0,Y 341.005,Z 302.821,A -85,B 0,C 180,E1 -14034.085,E2 -14034.085} C_VEL
LIN {X 0,Y 341.115,Z 302.804,A -85,B 0,C 180,E1 -14037.638,E2 -14037.638} C_VEL
LIN {X 0,Y 341.077,Z 302.808,A -85,B 0,C 180,E1 -14041.181,E2 -14041.181} C_VEL
LIN {X 0,Y 341.108,Z 302.805,A -85,B 0,C 180,E1 -14042.362,E2 -14042.362} C_VEL
LIN {X 0,Y 341.004,Z 302.821,A -85,B 0,C 180,E1 -14045.915,E2 -14045.915} C_VEL
LIN {X 0,Y 340.956,Z 302.825,A -85,B 0,C 180,E1 -14048.356,E2 -14048.356} C_VEL
LIN {X 0,Y 340.835,Z 302.841,A -85,B 0,C 180,E1 -14051.9,E2 -14051.9} C_VEL
LIN {X 0,Y 340.784,Z 302.848,A -85,B 0,C 180,E1 -14055.551,E2 -14055.551} C_VEL
LIN {X 0,Y 340.695,Z 302.859,A -85,B 0,C 180,E1 -14059.272,E2 -14059.272} C_VEL
LIN {X 0,Y 340.692,Z 302.856,A -85,B 0,C 180,E1 -14063.075,E2 -14063.075} C_VEL
LIN {X 0,Y 340.702,Z 302.858,A -85,B 0,C 180,E1 -14066.989,E2 -14066.989} C_VEL
LIN {X 0,Y 340.686,Z 302.859,A -85,B 0,C 180,E1 -14071.046,E2 -14071.046} C_VEL
LIN {X 0,Y 340.709,Z 302.857,A -85,B 0,C 180,E1 -14075.28,E2 -14075.28} C_VEL
LIN {X 0,Y 340.687,Z 302.852,A -85,B 0,C 180,E1 -14078.383,E2 -14078.383} C_VEL
LIN {X 0,Y 340.684,Z 302.856,A -85,B 0,C 180,E1 -14082.044,E2 -14082.044} C_VEL
LIN {X 0,Y 340.644,Z 302.863,A -85,B 0,C 180,E1 -14086.228,E2 -14086.228} C_VEL
LIN {X 0,Y 340.663,Z 302.86,A -85,B 0,C 180,E1 -14088.688,E2 -14088.688} C_VEL
LIN {X 0,Y 340.714,Z 302.854,A -85,B 0,C 180,E1 -14091.771,E2 -14091.771} C_VEL
LIN {X 0,Y 340.719,Z 302.852,A -85,B 0,C 180,E1 -14095.596,E2 -14095.596} C_VEL
LIN {X 0,Y 340.69,Z 302.858,A -85,B 0,C 180,E1 -14098.955,E2 -14098.955} C_VEL
LIN {X 0,Y 340.709,Z 302.849,A -85,B 0,C 180,E1 -14103.013,E2 -14103.013} C_VEL
LIN {X 0,Y 340.797,Z 303.106,A -85,B 0,C 180,E1 -14104.789,E2 -14104.789} C_VEL
LIN {X 0,Y 342.248,Z 311.048,A -85,B 0,C 180,E1 -14107.528,E2 -14107.528} C_VEL
LIN {X 0,Y 342.478,Z 315.399,A -85,B 0,C 180,E1 -14108.954,E2 -14108.954} C_VEL
LIN {X 0,Y 341.805,Z 323.774,A -85,B 0,C 180,E1 -14111.515,E2 -14111.515} C_VEL
LIN {X 0,Y 342.728,Z 329.073,A -85,B 0,C 180,E1 -14111.734,E2 -14111.734} C_VEL
LIN {X 0,Y 346.231,Z 351.034,A -85,B 0,C 180,E1 -14112.394,E2 -14112.394} C_VEL
LIN {X 0,Y 345.581,Z 399.96,A -85,B 0,C 180,E1 -14113.436,E2 -14113.436} C_VEL
LIN {X 0,Y 345.169,Z 409.434,A -85,B 0,C 180,E1 -14113.78,E2 -14113.78} C_VEL
LIN {X 0,Y 344.655,Z 419.441,A -85,B 0,C 180,E1 -14114.325,E2 -14114.325} C_VEL
LIN {X 0,Y 343.793,Z 430.806,A -85,B 0,C 180,E1 -14115.195,E2 -14115.195} C_VEL
LIN {X 0,Y 343.032,Z 439.37,A -85,B 0,C 180,E1 -14116.071,E2 -14116.071} C_VEL
LIN {X 0,Y 342.265,Z 447.427,A -85,B 0,C 180,E1 -14117.097,E2 -14117.097} C_VEL
LIN {X 0,Y 341.612,Z 454.081,A -85,B 0,C 180,E1 -14118.128,E2 -14118.128} C_VEL
LIN {X 0,Y 340.925,Z 460.396,A -85,B 0,C 180,E1 -14119.308,E2 -14119.308} C_VEL
LIN {X 0,Y 340.337,Z 465.641,A -85,B 0,C 180,E1 -14120.491,E2 -14120.491} C_VEL
LIN {X 0,Y 339.93,Z 470.015,A -85,B 0,C 180,E1 -14121.679,E2 -14121.679} C_VEL
LIN {X 0,Y 339.47,Z 475.171,A -85,B 0,C 180,E1 -14123.463,E2 -14123.463} C_VEL
LIN {X 0,Y 339.258,Z 478.953,A -85,B 0,C 180,E1 -14125.247,E2 -14125.247} C_VEL
LIN {X 0,Y 339.116,Z 480.691,A -85,B 0,C 180,E1 -14126.436,E2 -14126.436} C_VEL
LIN {X 0,Y 339.005,Z 481.934,A -85,B 0,C 180,E1 -14127.624,E2 -14127.624} C_VEL
LIN {X 0,Y 338.964,Z 482.708,A -85,B 0,C 180,E1 -14128.812,E2 -14128.812} C_VEL
LIN {X 0,Y 338.948,Z 483,A -85,B 0,C 180,E1 -14130,E2 -14130} C_VEL
LIN {X 0,Y 338.964,Z 482.703,A -85,B 0,C 180,E1 -14131.188,E2 -14131.188} C_VEL
LIN {X 0,Y 339.005,Z 481.921,A -85,B 0,C 180,E1 -14132.376,E2 -14132.376} C_VEL
LIN {X 0,Y 339.116,Z 480.668,A -85,B 0,C 180,E1 -14133.564,E2 -14133.564} C_VEL
LIN {X 0,Y 339.297,Z 477.771,A -85,B 0,C 180,E1 -14135.348,E2 -14135.348} C_VEL
LIN {X 0,Y 339.471,Z 475.434,A -85,B 0,C 180,E1 -14136.418,E2 -14136.418} C_VEL
LIN {X 0,Y 339.782,Z 471.873,A -85,B 0,C 180,E1 -14137.726,E2 -14137.726} C_VEL
LIN {X 0,Y 340.252,Z 466.746,A -85,B 0,C 180,E1 -14139.211,E2 -14139.211} C_VEL
LIN {X 0,Y 340.778,Z 461.733,A -85,B 0,C 180,E1 -14140.396,E2 -14140.396} C_VEL
LIN {X 0,Y 341.413,Z 455.694,A -85,B 0,C 180,E1 -14141.578,E2 -14141.578} C_VEL
LIN {X 0,Y 342.211,Z 448.343,A -85,B 0,C 180,E1 -14142.754,E2 -14142.754} C_VEL
LIN {X 0,Y 342.91,Z 440.467,A -85,B 0,C 180,E1 -14143.783,E2 -14143.783} C_VEL
LIN {X 0,Y 343.687,Z 432.142,A -85,B 0,C 180,E1 -14144.658,E2 -14144.658} C_VEL
LIN {X 0,Y 344.494,Z 421.5,A -85,B 0,C 180,E1 -14145.531,E2 -14145.531} C_VEL
LIN {X 0,Y 345.128,Z 409.899,A -85,B 0,C 180,E1 -14146.184,E2 -14146.184} C_VEL
LIN {X 0,Y 345.538,Z 400.162,A -85,B 0,C 180,E1 -14146.543,E2 -14146.543} C_VEL
LIN {X 0,Y 346.118,Z 349.564,A -85,B 0,C 180,E1 -14147.626,E2 -14147.626} C_VEL
LIN {X 0,Y 341.83,Z 324.131,A -85,B 0,C 180,E1 -14148.429,E2 -14148.429} C_VEL
LIN {X 0,Y 341.834,Z 322.477,A -85,B 0,C 180,E1 -14148.796,E2 -14148.796} C_VEL
LIN {X 0,Y 342.472,Z 315.341,A -85,B 0,C 180,E1 -14151.046,E2 -14151.046} C_VEL
LIN {X 0,Y 342.241,Z 311,A -85,B 0,C 180,E1 -14152.469,E2 -14152.469} C_VEL
LIN {X 0,Y 340.793,Z 302.964,A -85,B 0,C 180,E1 -14155.267,E2 -14155.267} C_VEL
LIN {X 0,Y 340.679,Z 302.859,A -85,B 0,C 180,E1 -14158.324,E2 -14158.324} C_VEL
LIN {X 0,Y 340.69,Z 302.858,A -85,B 0,C 180,E1 -14161.045,E2 -14161.045} C_VEL
LIN {X 0,Y 340.714,Z 302.856,A -85,B 0,C 180,E1 -14165.278,E2 -14165.278} C_VEL
LIN {X 0,Y 340.689,Z 302.857,A -85,B 0,C 180,E1 -14168.382,E2 -14168.382} C_VEL
LIN {X 0,Y 340.685,Z 302.854,A -85,B 0,C 180,E1 -14172.043,E2 -14172.043} C_VEL
LIN {X 0,Y 340.644,Z 302.863,A -85,B 0,C 180,E1 -14176.227,E2 -14176.227} C_VEL
LIN {X 0,Y 340.662,Z 302.861,A -85,B 0,C 180,E1 -14178.687,E2 -14178.687} C_VEL
LIN {X 0,Y 340.712,Z 302.849,A -85,B 0,C 180,E1 -14181.77,E2 -14181.77} C_VEL
LIN {X 0,Y 340.715,Z 302.854,A -85,B 0,C 180,E1 -14185.595,E2 -14185.595} C_VEL
LIN {X 0,Y 340.686,Z 302.86,A -85,B 0,C 180,E1 -14188.954,E2 -14188.954} C_VEL
LIN {X 0,Y 340.702,Z 302.858,A -85,B 0,C 180,E1 -14193.011,E2 -14193.011} C_VEL
LIN {X 0,Y 340.692,Z 302.856,A -85,B 0,C 180,E1 -14196.925,E2 -14196.925} C_VEL
LIN {X 0,Y 340.695,Z 302.859,A -85,B 0,C 180,E1 -14200.728,E2 -14200.728} C_VEL
LIN {X 0,Y 340.784,Z 302.848,A -85,B 0,C 180,E1 -14204.449,E2 -14204.449} C_VEL
LIN {X 0,Y 340.839,Z 302.84,A -85,B 0,C 180,E1 -14208.101,E2 -14208.101} C_VEL
LIN {X 0,Y 340.972,Z 302.823,A -85,B 0,C 180,E1 -14211.704,E2 -14211.704} C_VEL
LIN {X 0,Y 341.005,Z 302.821,A -85,B 0,C 180,E1 -14214.085,E2 -14214.085} C_VEL
LIN {X 0,Y 341.114,Z 302.804,A -85,B 0,C 180,E1 -14217.639,E2 -14217.639} C_VEL
LIN {X 0,Y 341.077,Z 302.808,A -85,B 0,C 180,E1 -14221.181,E2 -14221.181} C_VEL
LIN {X 0,Y 341.108,Z 302.805,A -85,B 0,C 180,E1 -14222.362,E2 -14222.362} C_VEL
LIN {X 0,Y 340.981,Z 302.82,A -85,B 0,C 180,E1 -14226.465,E2 -14226.465} C_VEL
LIN {X 0,Y 340.871,Z 302.837,A -85,B 0,C 180,E1 -14229.494,E2 -14229.494} C_VEL
LIN {X 0,Y 340.832,Z 302.838,A -85,B 0,C 180,E1 -14233.11,E2 -14233.11} C_VEL
LIN {X 0,Y 340.731,Z 302.851,A -85,B 0,C 180,E1 -14236.784,E2 -14236.784} C_VEL
LIN {X 0,Y 340.696,Z 302.859,A -85,B 0,C 180,E1 -14239.272,E2 -14239.272} C_VEL
LIN {X 0,Y 340.693,Z 302.856,A -85,B 0,C 180,E1 -14243.076,E2 -14243.076} C_VEL
LIN {X 0,Y 340.702,Z 302.857,A -85,B 0,C 180,E1 -14246.989,E2 -14246.989} C_VEL
LIN {X 0,Y 340.686,Z 302.859,A -85,B 0,C 180,E1 -14251.046,E2 -14251.046} C_VEL
LIN {X 0,Y 340.71,Z 302.857,A -85,B 0,C 180,E1 -14255.28,E2 -14255.28} C_VEL
LIN {X 0,Y 340.687,Z 302.853,A -85,B 0,C 180,E1 -14258.383,E2 -14258.383} C_VEL
LIN {X 0,Y 340.685,Z 302.856,A -85,B 0,C 180,E1 -14262.044,E2 -14262.044} C_VEL
LIN {X 0,Y 340.645,Z 302.862,A -85,B 0,C 180,E1 -14266.228,E2 -14266.228} C_VEL
LIN {X 0,Y 340.665,Z 302.861,A -85,B 0,C 180,E1 -14268.688,E2 -14268.688} C_VEL
LIN {X 0,Y 340.716,Z 302.853,A -85,B 0,C 180,E1 -14271.771,E2 -14271.771} C_VEL
LIN {X 0,Y 340.721,Z 302.851,A -85,B 0,C 180,E1 -14275.596,E2 -14275.596} C_VEL
LIN {X 0,Y 340.69,Z 302.859,A -85,B 0,C 180,E1 -14278.955,E2 -14278.955} C_VEL
LIN {X 0,Y 340.71,Z 302.85,A -85,B 0,C 180,E1 -14283.013,E2 -14283.013} C_VEL
LIN {X 0,Y 340.786,Z 302.979,A -85,B 0,C 180,E1 -14284.794,E2 -14284.794} C_VEL
LIN {X 0,Y 342.394,Z 312.06,A -85,B 0,C 180,E1 -14287.931,E2 -14287.931} C_VEL
LIN {X 0,Y 342.347,Z 317.153,A -85,B 0,C 180,E1 -14289.575,E2 -14289.575} C_VEL
LIN {X 0,Y 341.812,Z 323.7,A -85,B 0,C 180,E1 -14291.564,E2 -14291.564} C_VEL
LIN {X 0,Y 342.358,Z 327.033,A -85,B 0,C 180,E1 -14291.732,E2 -14291.732} C_VEL
LIN {X 0,Y 346.222,Z 350.651,A -85,B 0,C 180,E1 -14292.447,E2 -14292.447} C_VEL
LIN {X 0,Y 345.535,Z 399.923,A -85,B 0,C 180,E1 -14293.494,E2 -14293.494} C_VEL
LIN {X 0,Y 345.186,Z 408.913,A -85,B 0,C 180,E1 -14293.819,E2 -14293.819} C_VEL
LIN {X 0,Y 344.674,Z 418.459,A -85,B 0,C 180,E1 -14294.326,E2 -14294.326} C_VEL
LIN {X 0,Y 344.007,Z 428.478,A -85,B 0,C 180,E1 -14295.053,E2 -14295.053} C_VEL
LIN {X 0,Y 343.118,Z 438.871,A -85,B 0,C 180,E1 -14296.074,E2 -14296.074} C_VEL
LIN {X 0,Y 342.306,Z 447.017,A -85,B 0,C 180,E1 -14297.099,E2 -14297.099} C_VEL
LIN {X 0,Y 341.645,Z 453.739,A -85,B 0,C 180,E1 -14298.129,E2 -14298.129} C_VEL
LIN {X 0,Y 340.927,Z 460.104,A -85,B 0,C 180,E1 -14299.308,E2 -14299.308} C_VEL
LIN {X 0,Y 340.287,Z 466.57,A -85,B 0,C 180,E1 -14300.79,E2 -14300.79} C_VEL
LIN {X 0,Y 339.813,Z 471.729,A -85,B 0,C 180,E1 -14302.274,E2 -14302.274} C_VEL
LIN {X 0,Y 339.361,Z 476.505,A -85,B 0,C 180,E1 -14304.057,E2 -14304.057} C_VEL
LIN {X 0,Y 339.272,Z 478.835,A -85,B 0,C 180,E1 -14305.247,E2 -14305.247} C_VEL
LIN {X 0,Y 339.12,Z 480.607,A -85,B 0,C 180,E1 -14306.436,E2 -14306.436} C_VEL
LIN {X 0,Y 339.007,Z 481.885,A -85,B 0,C 180,E1 -14307.624,E2 -14307.624} C_VEL
LIN {X 0,Y 338.965,Z 482.691,A -85,B 0,C 180,E1 -14308.812,E2 -14308.812} C_VEL
LIN {X 0,Y 338.949,Z 482.998,A -85,B 0,C 180,E1 -14310,E2 -14310} C_VEL
LIN {X 0,Y 338.961,Z 482.72,A -85,B 0,C 180,E1 -14311.188,E2 -14311.188} C_VEL
LIN {X 0,Y 338.994,Z 481.971,A -85,B 0,C 180,E1 -14312.376,E2 -14312.376} C_VEL
LIN {X 0,Y 339.112,Z 480.752,A -85,B 0,C 180,E1 -14313.565,E2 -14313.565} C_VEL
LIN {X 0,Y 339.291,Z 477.889,A -85,B 0,C 180,E1 -14315.348,E2 -14315.348} C_VEL
LIN {X 0,Y 339.533,Z 474.789,A -85,B 0,C 180,E1 -14316.732,E2 -14316.732} C_VEL
LIN {X 0,Y 339.921,Z 470.158,A -85,B 0,C 180,E1 -14318.321,E2 -14318.321} C_VEL
LIN {X 0,Y 340.482,Z 464.645,A -85,B 0,C 180,E1 -14319.804,E2 -14319.804} C_VEL
LIN {X 0,Y 341.255,Z 457.721,A -85,B 0,C 180,E1 -14321.282,E2 -14321.282} C_VEL
LIN {X 0,Y 342.071,Z 449.773,A -85,B 0,C 180,E1 -14322.609,E2 -14322.609} C_VEL
LIN {X 0,Y 342.786,Z 442.194,A -85,B 0,C 180,E1 -14323.637,E2 -14323.637} C_VEL
LIN {X 0,Y 343.594,Z 434.252,A -85,B 0,C 180,E1 -14324.511,E2 -14324.511} C_VEL
LIN {X 0,Y 344.239,Z 426.051,A -85,B 0,C 180,E1 -14325.239,E2 -14325.239} C_VEL
LIN {X 0,Y 344.783,Z 417.739,A -85,B 0,C 180,E1 -14325.821,E2 -14325.821} C_VEL
LIN {X 0,Y 345.199,Z 408.756,A -85,B 0,C 180,E1 -14326.294,E2 -14326.294} C_VEL
LIN {X 0,Y 345.576,Z 399.662,A -85,B 0,C 180,E1 -14326.618,E2 -14326.618} C_VEL
LIN {X 0,Y 346.174,Z 350.013,A -85,B 0,C 180,E1 -14327.676,E2 -14327.676} C_VEL
LIN {X 0,Y 342.032,Z 325.282,A -85,B 0,C 180,E1 -14328.437,E2 -14328.437} C_VEL
LIN {X 0,Y 341.781,Z 323.474,A -85,B 0,C 180,E1 -14328.585,E2 -14328.585} C_VEL
LIN {X 0,Y 342.461,Z 315.538,A -85,B 0,C 180,E1 -14331.047,E2 -14331.047} C_VEL
LIN {X 0,Y 342.249,Z 311.187,A -85,B 0,C 180,E1 -14332.472,E2 -14332.472} C_VEL
LIN {X 0,Y 340.829,Z 303.276,A -85,B 0,C 180,E1 -14335.191,E2 -14335.191} C_VEL
LIN {X 0,Y 340.196,Z 302.912,A -85,B 0,C 180,E1 -14335.802,E2 -14335.802} C_VEL
LIN {X 0,Y 336.89,Z 303.33,A -85,B 0,C 180,E1 -14337.714,E2 -14337.714} C_VEL
LIN {X 0,Y 334.694,Z 303.777,A -85,B 0,C 180,E1 -14339.045,E2 -14339.045} C_VEL
LIN {X 0,Y 333.651,Z 303.733,A -85,B 0,C 180,E1 -14340.42,E2 -14340.42} C_VEL
LIN {X 0,Y 333.635,Z 303.74,A -85,B 0,C 180,E1 -14343.208,E2 -14343.208} C_VEL
LIN {X 0,Y 333.672,Z 303.73,A -85,B 0,C 180,E1 -14346.138,E2 -14346.138} C_VEL
LIN {X 0,Y 333.616,Z 303.742,A -85,B 0,C 180,E1 -14349.195,E2 -14349.195} C_VEL
LIN {X 0,Y 333.622,Z 303.733,A -85,B 0,C 180,E1 -14352.498,E2 -14352.498} C_VEL
LIN {X 0,Y 333.589,Z 303.742,A -85,B 0,C 180,E1 -14355.954,E2 -14355.954} C_VEL
LIN {X 0,Y 333.597,Z 303.737,A -85,B 0,C 180,E1 -14359.324,E2 -14359.324} C_VEL
LIN {X 0,Y 333.656,Z 303.734,A -85,B 0,C 180,E1 -14363.168,E2 -14363.168} C_VEL
LIN {X 0,Y 333.667,Z 303.733,A -85,B 0,C 180,E1 -14365.34,E2 -14365.34} C_VEL
LIN {X 0,Y 333.623,Z 303.738,A -85,B 0,C 180,E1 -14368.221,E2 -14368.221} C_VEL
LIN {X 0,Y 333.645,Z 303.736,A -85,B 0,C 180,E1 -14371.021,E2 -14371.021} C_VEL
LIN {X 0,Y 333.656,Z 303.734,A -85,B 0,C 180,E1 -14375.085,E2 -14375.085} C_VEL
LIN {X 0,Y 333.644,Z 303.735,A -85,B 0,C 180,E1 -14379.017,E2 -14379.017} C_VEL
LIN {X 0,Y 333.704,Z 303.727,A -85,B 0,C 180,E1 -14381.584,E2 -14381.584} C_VEL
LIN {X 0,Y 333.766,Z 303.717,A -85,B 0,C 180,E1 -14385.6,E2 -14385.6} C_VEL
LIN {X 0,Y 333.809,Z 303.714,A -85,B 0,C 180,E1 -14389.077,E2 -14389.077} C_VEL
LIN {X 0,Y 333.948,Z 303.696,A -85,B 0,C 180,E1 -14392.746,E2 -14392.746} C_VEL
LIN {X 0,Y 333.767,Z 303.715,A -85,B 0,C 180,E1 -14395.168,E2 -14395.168} C_VEL
LIN {X 0,Y 334.055,Z 303.683,A -85,B 0,C 180,E1 -14397.588,E2 -14397.588} C_VEL
LIN {X 0,Y 334.048,Z 303.684,A -85,B 0,C 180,E1 -14401.205,E2 -14401.205} C_VEL
LIN {X 0,Y 334.048,Z 303.684,A -85,B 0,C 180,E1 -14402.411,E2 -14402.411} C_VEL
LIN {X 0,Y 333.978,Z 303.695,A -85,B 0,C 180,E1 -14406.04,E2 -14406.04} C_VEL
LIN {X 0,Y 333.905,Z 303.702,A -85,B 0,C 180,E1 -14408.472,E2 -14408.472} C_VEL
LIN {X 0,Y 333.777,Z 303.717,A -85,B 0,C 180,E1 -14412.155,E2 -14412.155} C_VEL
LIN {X 0,Y 333.709,Z 303.729,A -85,B 0,C 180,E1 -14415.889,E2 -14415.889} C_VEL
LIN {X 0,Y 333.687,Z 303.729,A -85,B 0,C 180,E1 -14418.603,E2 -14418.603} C_VEL
LIN {X 0,Y 333.641,Z 303.732,A -85,B 0,C 180,E1 -14422.282,E2 -14422.282} C_VEL
LIN {X 0,Y 333.65,Z 303.736,A -85,B 0,C 180,E1 -14425.078,E2 -14425.078} C_VEL
LIN {X 0,Y 333.644,Z 303.736,A -85,B 0,C 180,E1 -14428.978,E2 -14428.978} C_VEL
LIN {X 0,Y 333.637,Z 303.736,A -85,B 0,C 180,E1 -14432.587,E2 -14432.587} C_VEL
LIN {X 0,Y 333.667,Z 303.729,A -85,B 0,C 180,E1 -14436.14,E2 -14436.14} C_VEL
LIN {X 0,Y 333.595,Z 303.736,A -85,B 0,C 180,E1 -14439.199,E2 -14439.199} C_VEL
LIN {X 0,Y 333.62,Z 303.737,A -85,B 0,C 180,E1 -14442.499,E2 -14442.499} C_VEL
LIN {X 0,Y 333.588,Z 303.741,A -85,B 0,C 180,E1 -14445.955,E2 -14445.955} C_VEL
LIN {X 0,Y 333.597,Z 303.739,A -85,B 0,C 180,E1 -14449.325,E2 -14449.325} C_VEL
LIN {X 0,Y 333.658,Z 303.733,A -85,B 0,C 180,E1 -14453.169,E2 -14453.169} C_VEL
LIN {X 0,Y 333.67,Z 303.73,A -85,B 0,C 180,E1 -14455.342,E2 -14455.342} C_VEL
LIN {X 0,Y 333.626,Z 303.74,A -85,B 0,C 180,E1 -14458.222,E2 -14458.222} C_VEL
LIN {X 0,Y 333.648,Z 303.736,A -85,B 0,C 180,E1 -14461.023,E2 -14461.023} C_VEL
LIN {X 0,Y 333.733,Z 303.845,A -85,B 0,C 180,E1 -14464.447,E2 -14464.447} C_VEL
LIN {X 0,Y 335.206,Z 311.849,A -85,B 0,C 180,E1 -14467.296,E2 -14467.296} C_VEL
LIN {X 0,Y 335.435,Z 317.352,A -85,B 0,C 180,E1 -14469.135,E2 -14469.135} C_VEL
LIN {X 0,Y 334.864,Z 323.625,A -85,B 0,C 180,E1 -14471.095,E2 -14471.095} C_VEL
LIN {X 0,Y 335.404,Z 326.86,A -85,B 0,C 180,E1 -14471.271,E2 -14471.271} C_VEL
LIN {X 0,Y 339.427,Z 350.541,A -85,B 0,C 180,E1 -14472.018,E2 -14472.018} C_VEL
LIN {X 0,Y 338.787,Z 399.287,A -85,B 0,C 180,E1 -14473.073,E2 -14473.073} C_VEL
LIN {X 0,Y 338.387,Z 408.612,A -85,B 0,C 180,E1 -14473.407,E2 -14473.407} C_VEL
LIN {X 0,Y 337.869,Z 418.238,A -85,B 0,C 180,E1 -14473.924,E2 -14473.924} C_VEL
LIN {X 0,Y 337.271,Z 427.373,A -85,B 0,C 180,E1 -14474.593,E2 -14474.593} C_VEL
LIN {X 0,Y 336.313,Z 438.143,A -85,B 0,C 180,E1 -14475.632,E2 -14475.632} C_VEL
LIN {X 0,Y 335.432,Z 446.409,A -85,B 0,C 180,E1 -14476.675,E2 -14476.675} C_VEL
LIN {X 0,Y 334.657,Z 454.083,A -85,B 0,C 180,E1 -14477.878,E2 -14477.878} C_VEL
LIN {X 0,Y 333.941,Z 460.398,A -85,B 0,C 180,E1 -14479.082,E2 -14479.082} C_VEL
LIN {X 0,Y 333.335,Z 465.643,A -85,B 0,C 180,E1 -14480.29,E2 -14480.29} C_VEL
LIN {X 0,Y 332.896,Z 470.016,A -85,B 0,C 180,E1 -14481.502,E2 -14481.502} C_VEL
LIN {X 0,Y 332.592,Z 473.654,A -85,B 0,C 180,E1 -14482.716,E2 -14482.716} C_VEL
LIN {X 0,Y 332.307,Z 476.639,A -85,B 0,C 180,E1 -14483.93,E2 -14483.93} C_VEL
LIN {X 0,Y 332.183,Z 478.954,A -85,B 0,C 180,E1 -14485.145,E2 -14485.145} C_VEL
LIN {X 0,Y 332.048,Z 480.691,A -85,B 0,C 180,E1 -14486.36,E2 -14486.36} C_VEL
LIN {X 0,Y 331.924,Z 481.935,A -85,B 0,C 180,E1 -14487.573,E2 -14487.573} C_VEL
LIN {X 0,Y 331.873,Z 482.708,A -85,B 0,C 180,E1 -14488.787,E2 -14488.787} C_VEL
LIN {X 0,Y 331.855,Z 483,A -85,B 0,C 180,E1 -14490,E2 -14490} C_VEL
LIN {X 0,Y 331.873,Z 482.703,A -85,B 0,C 180,E1 -14491.213,E2 -14491.213} C_VEL
LIN {X 0,Y 331.924,Z 481.921,A -85,B 0,C 180,E1 -14492.427,E2 -14492.427} C_VEL
LIN {X 0,Y 332.047,Z 480.668,A -85,B 0,C 180,E1 -14493.64,E2 -14493.64} C_VEL
LIN {X 0,Y 332.208,Z 477.77,A -85,B 0,C 180,E1 -14495.463,E2 -14495.463} C_VEL
LIN {X 0,Y 332.421,Z 475.28,A -85,B 0,C 180,E1 -14496.616,E2 -14496.616} C_VEL
LIN {X 0,Y 332.892,Z 469.959,A -85,B 0,C 180,E1 -14498.498,E2 -14498.498} C_VEL
LIN {X 0,Y 333.632,Z 463.144,A -85,B 0,C 180,E1 -14500.314,E2 -14500.314} C_VEL
LIN {X 0,Y 334.449,Z 455.692,A -85,B 0,C 180,E1 -14501.822,E2 -14501.822} C_VEL
LIN {X 0,Y 335.269,Z 448.34,A -85,B 0,C 180,E1 -14503.023,E2 -14503.023} C_VEL
LIN {X 0,Y 336.005,Z 440.464,A -85,B 0,C 180,E1 -14504.072,E2 -14504.072} C_VEL
LIN {X 0,Y 336.84,Z 432.137,A -85,B 0,C 180,E1 -14504.963,E2 -14504.963} C_VEL
LIN {X 0,Y 337.667,Z 421.494,A -85,B 0,C 180,E1 -14505.853,E2 -14505.853} C_VEL
LIN {X 0,Y 338.325,Z 409.89,A -85,B 0,C 180,E1 -14506.518,E2 -14506.518} C_VEL
LIN {X 0,Y 338.704,Z 401.445,A -85,B 0,C 180,E1 -14506.848,E2 -14506.848} C_VEL
LIN {X 0,Y 339.118,Z 376.963,A -85,B 0,C 180,E1 -14507.405,E2 -14507.405} C_VEL
LIN {X 0,Y 339.357,Z 350.525,A -85,B 0,C 180,E1 -14507.968,E2 -14507.968} C_VEL
LIN {X 0,Y 335.077,Z 325.266,A -85,B 0,C 180,E1 -14508.77,E2 -14508.77} C_VEL
LIN {X 0,Y 334.856,Z 323.761,A -85,B 0,C 180,E1 -14508.867,E2 -14508.867} C_VEL
LIN {X 0,Y 335.429,Z 317.291,A -85,B 0,C 180,E1 -14510.866,E2 -14510.866} C_VEL
LIN {X 0,Y 335.427,Z 313.387,A -85,B 0,C 180,E1 -14512.156,E2 -14512.156} C_VEL
LIN {X 0,Y 333.901,Z 304.777,A -85,B 0,C 180,E1 -14515.168,E2 -14515.168} C_VEL
LIN {X 0,Y 333.721,Z 303.796,A -85,B 0,C 180,E1 -14515.631,E2 -14515.631} C_VEL
LIN {X 0,Y 333.65,Z 303.736,A -85,B 0,C 180,E1 -14518.977,E2 -14518.977} C_VEL
LIN {X 0,Y 333.64,Z 303.736,A -85,B 0,C 180,E1 -14522.586,E2 -14522.586} C_VEL
LIN {X 0,Y 333.671,Z 303.731,A -85,B 0,C 180,E1 -14526.139,E2 -14526.139} C_VEL
LIN {X 0,Y 333.615,Z 303.742,A -85,B 0,C 180,E1 -14529.196,E2 -14529.196} C_VEL
LIN {X 0,Y 333.621,Z 303.734,A -85,B 0,C 180,E1 -14532.498,E2 -14532.498} C_VEL
LIN {X 0,Y 333.588,Z 303.742,A -85,B 0,C 180,E1 -14535.954,E2 -14535.954} C_VEL
LIN {X 0,Y 333.596,Z 303.737,A -85,B 0,C 180,E1 -14539.324,E2 -14539.324} C_VEL
LIN {X 0,Y 333.655,Z 303.734,A -85,B 0,C 180,E1 -14543.168,E2 -14543.168} C_VEL
LIN {X 0,Y 333.666,Z 303.733,A -85,B 0,C 180,E1 -14545.341,E2 -14545.341} C_VEL
LIN {X 0,Y 333.622,Z 303.738,A -85,B 0,C 180,E1 -14548.221,E2 -14548.221} C_VEL
LIN {X 0,Y 333.644,Z 303.736,A -85,B 0,C 180,E1 -14551.022,E2 -14551.022} C_VEL
LIN {X 0,Y 333.655,Z 303.734,A -85,B 0,C 180,E1 -14555.085,E2 -14555.085} C_VEL
LIN {X 0,Y 333.643,Z 303.735,A -85,B 0,C 180,E1 -14559.017,E2 -14559.017} C_VEL
LIN {X 0,Y 333.703,Z 303.727,A -85,B 0,C 180,E1 -14561.584,E2 -14561.584} C_VEL
LIN {X 0,Y 333.766,Z 303.717,A -85,B 0,C 180,E1 -14565.6,E2 -14565.6} C_VEL
LIN {X 0,Y 333.808,Z 303.714,A -85,B 0,C 180,E1 -14569.077,E2 -14569.077} C_VEL
LIN {X 0,Y 333.947,Z 303.696,A -85,B 0,C 180,E1 -14572.746,E2 -14572.746} C_VEL
LIN {X 0,Y 333.767,Z 303.715,A -85,B 0,C 180,E1 -14575.169,E2 -14575.169} C_VEL
LIN {X 0,Y 334.055,Z 303.683,A -85,B 0,C 180,E1 -14577.589,E2 -14577.589} C_VEL
LIN {X 0,Y 334.048,Z 303.684,A -85,B 0,C 180,E1 -14581.206,E2 -14581.206} C_VEL
LIN {X 0,Y 334.048,Z 303.684,A -85,B 0,C 180,E1 -14582.412,E2 -14582.412} C_VEL
LIN {X 0,Y 333.951,Z 303.696,A -85,B 0,C 180,E1 -14586.456,E2 -14586.456} C_VEL
LIN {X 0,Y 333.81,Z 303.718,A -85,B 0,C 180,E1 -14589.697,E2 -14589.697} C_VEL
LIN {X 0,Y 333.777,Z 303.718,A -85,B 0,C 180,E1 -14593.392,E2 -14593.392} C_VEL
LIN {X 0,Y 333.676,Z 303.732,A -85,B 0,C 180,E1 -14597.15,E2 -14597.15} C_VEL
LIN {X 0,Y 333.64,Z 303.738,A -85,B 0,C 180,E1 -14599.696,E2 -14599.696} C_VEL
LIN {X 0,Y 333.642,Z 303.731,A -85,B 0,C 180,E1 -14602.282,E2 -14602.282} C_VEL
LIN {X 0,Y 333.649,Z 303.736,A -85,B 0,C 180,E1 -14605.078,E2 -14605.078} C_VEL
LIN {X 0,Y 333.642,Z 303.736,A -85,B 0,C 180,E1 -14608.979,E2 -14608.979} C_VEL
LIN {X 0,Y 333.638,Z 303.736,A -85,B 0,C 180,E1 -14612.587,E2 -14612.587} C_VEL
LIN {X 0,Y 333.667,Z 303.729,A -85,B 0,C 180,E1 -14616.14,E2 -14616.14} C_VEL
LIN {X 0,Y 333.596,Z 303.736,A -85,B 0,C 180,E1 -14619.2,E2 -14619.2} C_VEL
LIN {X 0,Y 333.621,Z 303.737,A -85,B 0,C 180,E1 -14622.499,E2 -14622.499} C_VEL
LIN {X 0,Y 333.589,Z 303.741,A -85,B 0,C 180,E1 -14625.955,E2 -14625.955} C_VEL
LIN {X 0,Y 333.598,Z 303.738,A -85,B 0,C 180,E1 -14629.325,E2 -14629.325} C_VEL
LIN {X 0,Y 333.66,Z 303.734,A -85,B 0,C 180,E1 -14633.169,E2 -14633.169} C_VEL
LIN {X 0,Y 333.671,Z 303.73,A -85,B 0,C 180,E1 -14635.342,E2 -14635.342} C_VEL
LIN {X 0,Y 333.627,Z 303.739,A -85,B 0,C 180,E1 -14638.222,E2 -14638.222} C_VEL
LIN {X 0,Y 333.627,Z 303.739,A -85,B 0,C 180,E1 -14641.021,E2 -14641.021} C_VEL
LIN {X 0,Y 333.738,Z 303.867,A -85,B 0,C 180,E1 -14644.528,E2 -14644.528} C_VEL
LIN {X 0,Y 335.192,Z 311.675,A -85,B 0,C 180,E1 -14647.302,E2 -14647.302} C_VEL
LIN {X 0,Y 335.5,Z 315.203,A -85,B 0,C 180,E1 -14648.495,E2 -14648.495} C_VEL
LIN {X 0,Y 334.882,Z 322.874,A -85,B 0,C 180,E1 -14650.964,E2 -14650.964} C_VEL
LIN {X 0,Y 334.918,Z 324.272,A -85,B 0,C 180,E1 -14651.229,E2 -14651.229} C_VEL
LIN {X 0,Y 339.417,Z 350.875,A -85,B 0,C 180,E1 -14652.088,E2 -14652.088} C_VEL
LIN {X 0,Y 338.745,Z 399.941,A -85,B 0,C 180,E1 -14653.154,E2 -14653.154} C_VEL
LIN {X 0,Y 338.343,Z 409.756,A -85,B 0,C 180,E1 -14653.521,E2 -14653.521} C_VEL
LIN {X 0,Y 337.7,Z 420.866,A -85,B 0,C 180,E1 -14654.149,E2 -14654.149} C_VEL
LIN {X 0,Y 336.885,Z 431.701,A -85,B 0,C 180,E1 -14655.039,E2 -14655.039} C_VEL
LIN {X 0,Y 336.085,Z 440.105,A -85,B 0,C 180,E1 -14655.931,E2 -14655.931} C_VEL
LIN {X 0,Y 335.285,Z 448.042,A -85,B 0,C 180,E1 -14656.978,E2 -14656.978} C_VEL
LIN {X 0,Y 334.709,Z 453.742,A -85,B 0,C 180,E1 -14657.88,E2 -14657.88} C_VEL
LIN {X 0,Y 333.948,Z 460.107,A -85,B 0,C 180,E1 -14659.082,E2 -14659.082} C_VEL
LIN {X 0,Y 333.265,Z 466.572,A -85,B 0,C 180,E1 -14660.594,E2 -14660.594} C_VEL
LIN {X 0,Y 332.757,Z 471.731,A -85,B 0,C 180,E1 -14662.11,E2 -14662.11} C_VEL
LIN {X 0,Y 332.309,Z 476.506,A -85,B 0,C 180,E1 -14663.93,E2 -14663.93} C_VEL
LIN {X 0,Y 332.194,Z 478.836,A -85,B 0,C 180,E1 -14665.146,E2 -14665.146} C_VEL
LIN {X 0,Y 332.052,Z 480.608,A -85,B 0,C 180,E1 -14666.36,E2 -14666.36} C_VEL
LIN {X 0,Y 331.925,Z 481.885,A -85,B 0,C 180,E1 -14667.573,E2 -14667.573} C_VEL
LIN {X 0,Y 331.875,Z 482.691,A -85,B 0,C 180,E1 -14668.787,E2 -14668.787} C_VEL
LIN {X 0,Y 331.856,Z 482.998,A -85,B 0,C 180,E1 -14670,E2 -14670} C_VEL
LIN {X 0,Y 331.871,Z 482.72,A -85,B 0,C 180,E1 -14671.213,E2 -14671.213} C_VEL
LIN {X 0,Y 331.913,Z 481.97,A -85,B 0,C 180,E1 -14672.427,E2 -14672.427} C_VEL
LIN {X 0,Y 332.044,Z 480.751,A -85,B 0,C 180,E1 -14673.641,E2 -14673.641} C_VEL
LIN {X 0,Y 332.202,Z 477.888,A -85,B 0,C 180,E1 -14675.463,E2 -14675.463} C_VEL
LIN {X 0,Y 332.393,Z 475.435,A -85,B 0,C 180,E1 -14676.617,E2 -14676.617} C_VEL
LIN {X 0,Y 332.888,Z 470.157,A -85,B 0,C 180,E1 -14678.498,E2 -14678.498} C_VEL
LIN {X 0,Y 333.467,Z 464.643,A -85,B 0,C 180,E1 -14680.013,E2 -14680.013} C_VEL
LIN {X 0,Y 334.301,Z 457.719,A -85,B 0,C 180,E1 -14681.52,E2 -14681.52} C_VEL
LIN {X 0,Y 335.129,Z 449.769,A -85,B 0,C 180,E1 -14682.874,E2 -14682.874} C_VEL
LIN {X 0,Y 335.877,Z 442.19,A -85,B 0,C 180,E1 -14683.923,E2 -14683.923} C_VEL
LIN {X 0,Y 336.718,Z 434.247,A -85,B 0,C 180,E1 -14684.814,E2 -14684.814} C_VEL
LIN {X 0,Y 337.398,Z 426.044,A -85,B 0,C 180,E1 -14685.556,E2 -14685.556} C_VEL
LIN {X 0,Y 337.973,Z 417.731,A -85,B 0,C 180,E1 -14686.148,E2 -14686.148} C_VEL
LIN {X 0,Y 338.401,Z 408.745,A -85,B 0,C 180,E1 -14686.631,E2 -14686.631} C_VEL
LIN {X 0,Y 338.775,Z 399.793,A -85,B 0,C 180,E1 -14686.957,E2 -14686.957} C_VEL
LIN {X 0,Y 339.381,Z 350.488,A -85,B 0,C 180,E1 -14688.031,E2 -14688.031} C_VEL
LIN {X 0,Y 335.222,Z 325.852,A -85,B 0,C 180,E1 -14688.807,E2 -14688.807} C_VEL
LIN {X 0,Y 334.866,Z 323.658,A -85,B 0,C 180,E1 -14688.945,E2 -14688.945} C_VEL
LIN {X 0,Y 335.496,Z 315.537,A -85,B 0,C 180,E1 -14691.505,E2 -14691.505} C_VEL
LIN {X 0,Y 335.071,Z 311.089,A -85,B 0,C 180,E1 -14693.013,E2 -14693.013} C_VEL
LIN {X 0,Y 333.733,Z 303.817,A -85,B 0,C 180,E1 -14695.634,E2 -14695.634} C_VEL
LIN {X 0,Y 333.651,Z 303.735,A -85,B 0,C 180,E1 -14698.977,E2 -14698.977} C_VEL
LIN {X 0,Y 333.651,Z 303.733,A -85,B 0,C 180,E1 -14700.42,E2 -14700.42} C_VEL
LIN {X 0,Y 332.939,Z 303.825,A -85,B 0,C 180,E1 -14701.428,E2 -14701.428} C_VEL
LIN {X 0,Y 330.103,Z 304.178,A -85,B 0,C 180,E1 -14703.069,E2 -14703.069} C_VEL
LIN {X 0,Y 327.721,Z 304.477,A -85,B 0,C 180,E1 -14704.397,E2 -14704.397} C_VEL
LIN {X 0,Y 326.688,Z 304.602,A -85,B 0,C 180,E1 -14705.425,E2 -14705.425} C_VEL
LIN {X 0,Y 326.596,Z 304.612,A -85,B 0,C 180,E1 -14705.773,E2 -14705.773} C_VEL
LIN {X 0,Y 326.584,Z 304.617,A -85,B 0,C 180,E1 -14709.221,E2 -14709.221} C_VEL
LIN {X 0,Y 326.567,Z 304.614,A -85,B 0,C 180,E1 -14712.97,E2 -14712.97} C_VEL
LIN {X 0,Y 326.568,Z 304.621,A -85,B 0,C 180,E1 -14717.028,E2 -14717.028} C_VEL
LIN {X 0,Y 326.581,Z 304.608,A -85,B 0,C 180,E1 -14720.778,E2 -14720.778} C_VEL
LIN {X 0,Y 326.605,Z 304.61,A -85,B 0,C 180,E1 -14724.479,E2 -14724.479} C_VEL
LIN {X 0,Y 326.602,Z 304.612,A -85,B 0,C 180,E1 -14727.455,E2 -14727.455} C_VEL
LIN {X 0,Y 326.609,Z 304.61,A -85,B 0,C 180,E1 -14730.336,E2 -14730.336} C_VEL
LIN {X 0,Y 326.593,Z 304.617,A -85,B 0,C 180,E1 -14734.508,E2 -14734.508} C_VEL
LIN {X 0,Y 326.601,Z 304.612,A -85,B 0,C 180,E1 -14738.542,E2 -14738.542} C_VEL
LIN {X 0,Y 326.624,Z 304.614,A -85,B 0,C 180,E1 -14742.468,E2 -14742.468} C_VEL
LIN {X 0,Y 326.735,Z 304.595,A -85,B 0,C 180,E1 -14746.313,E2 -14746.313} C_VEL
LIN {X 0,Y 326.775,Z 304.593,A -85,B 0,C 180,E1 -14750.092,E2 -14750.092} C_VEL
LIN {X 0,Y 326.933,Z 304.571,A -85,B 0,C 180,E1 -14753.83,E2 -14753.83} C_VEL
LIN {X 0,Y 326.999,Z 304.561,A -85,B 0,C 180,E1 -14757.536,E2 -14757.536} C_VEL
LIN {X 0,Y 327.018,Z 304.56,A -85,B 0,C 180,E1 -14761.231,E2 -14761.231} C_VEL
LIN {X 0,Y 326.728,Z 304.597,A -85,B 0,C 180,E1 -14763.7,E2 -14763.7} C_VEL
LIN {X 0,Y 326.933,Z 304.572,A -85,B 0,C 180,E1 -14766.17,E2 -14766.17} C_VEL
LIN {X 0,Y 326.773,Z 304.594,A -85,B 0,C 180,E1 -14769.907,E2 -14769.907} C_VEL
LIN {X 0,Y 326.734,Z 304.595,A -85,B 0,C 180,E1 -14773.686,E2 -14773.686} C_VEL
LIN {X 0,Y 326.623,Z 304.614,A -85,B 0,C 180,E1 -14777.532,E2 -14777.532} C_VEL
LIN {X 0,Y 326.6,Z 304.613,A -85,B 0,C 180,E1 -14781.458,E2 -14781.458} C_VEL
LIN {X 0,Y 326.592,Z 304.618,A -85,B 0,C 180,E1 -14785.492,E2 -14785.492} C_VEL
LIN {X 0,Y 326.608,Z 304.611,A -85,B 0,C 180,E1 -14789.664,E2 -14789.664} C_VEL
LIN {X 0,Y 326.611,Z 304.614,A -85,B 0,C 180,E1 -14792.946,E2 -14792.946} C_VEL
LIN {X 0,Y 326.604,Z 304.611,A -85,B 0,C 180,E1 -14795.521,E2 -14795.521} C_VEL
LIN {X 0,Y 326.565,Z 304.61,A -85,B 0,C 180,E1 -14799.219,E2 -14799.219} C_VEL
LIN {X 0,Y 326.566,Z 304.62,A -85,B 0,C 180,E1 -14802.971,E2 -14802.971} C_VEL
LIN {X 0,Y 326.566,Z 304.614,A -85,B 0,C 180,E1 -14807.03,E2 -14807.03} C_VEL
LIN {X 0,Y 326.577,Z 304.616,A -85,B 0,C 180,E1 -14811.386,E2 -14811.386} C_VEL
LIN {X 0,Y 326.615,Z 304.61,A -85,B 0,C 180,E1 -14814.852,E2 -14814.852} C_VEL
LIN {X 0,Y 326.605,Z 304.612,A -85,B 0,C 180,E1 -14817.456,E2 -14817.456} C_VEL
LIN {X 0,Y 326.612,Z 304.614,A -85,B 0,C 180,E1 -14820.337,E2 -14820.337} C_VEL
LIN {X 0,Y 326.679,Z 304.744,A -85,B 0,C 180,E1 -14824.174,E2 -14824.174} C_VEL
LIN {X 0,Y 328.276,Z 313.45,A -85,B 0,C 180,E1 -14827.335,E2 -14827.335} C_VEL
LIN {X 0,Y 328.483,Z 317.354,A -85,B 0,C 180,E1 -14828.672,E2 -14828.672} C_VEL
LIN {X 0,Y 327.959,Z 323.784,A -85,B 0,C 180,E1 -14830.705,E2 -14830.705} C_VEL
LIN {X 0,Y 329.085,Z 329.8,A -85,B 0,C 180,E1 -14830.963,E2 -14830.963} C_VEL
LIN {X 0,Y 332.676,Z 351.35,A -85,B 0,C 180,E1 -14831.658,E2 -14831.658} C_VEL
LIN {X 0,Y 332.008,Z 399.39,A -85,B 0,C 180,E1 -14832.719,E2 -14832.719} C_VEL
LIN {X 0,Y 331.6,Z 408.621,A -85,B 0,C 180,E1 -14833.057,E2 -14833.057} C_VEL
LIN {X 0,Y 331.066,Z 418.245,A -85,B 0,C 180,E1 -14833.585,E2 -14833.585} C_VEL
LIN {X 0,Y 330.434,Z 427.378,A -85,B 0,C 180,E1 -14834.266,E2 -14834.266} C_VEL
LIN {X 0,Y 329.448,Z 438.147,A -85,B 0,C 180,E1 -14835.326,E2 -14835.326} C_VEL
LIN {X 0,Y 328.52,Z 446.412,A -85,B 0,C 180,E1 -14836.39,E2 -14836.39} C_VEL
LIN {X 0,Y 327.723,Z 454.086,A -85,B 0,C 180,E1 -14837.617,E2 -14837.617} C_VEL
LIN {X 0,Y 326.977,Z 460.4,A -85,B 0,C 180,E1 -14838.846,E2 -14838.846} C_VEL
LIN {X 0,Y 326.339,Z 465.645,A -85,B 0,C 180,E1 -14840.079,E2 -14840.079} C_VEL
LIN {X 0,Y 325.88,Z 470.017,A -85,B 0,C 180,E1 -14841.317,E2 -14841.317} C_VEL
LIN {X 0,Y 325.352,Z 475.174,A -85,B 0,C 180,E1 -14843.178,E2 -14843.178} C_VEL
LIN {X 0,Y 325.089,Z 478.955,A -85,B 0,C 180,E1 -14845.039,E2 -14845.039} C_VEL
LIN {X 0,Y 324.981,Z 480.692,A -85,B 0,C 180,E1 -14846.28,E2 -14846.28} C_VEL
LIN {X 0,Y 324.845,Z 481.935,A -85,B 0,C 180,E1 -14847.52,E2 -14847.52} C_VEL
LIN {X 0,Y 324.785,Z 482.708,A -85,B 0,C 180,E1 -14848.76,E2 -14848.76} C_VEL
LIN {X 0,Y 324.765,Z 483,A -85,B 0,C 180,E1 -14850,E2 -14850} C_VEL
LIN {X 0,Y 324.785,Z 482.703,A -85,B 0,C 180,E1 -14851.24,E2 -14851.24} C_VEL
LIN {X 0,Y 324.845,Z 481.92,A -85,B 0,C 180,E1 -14852.48,E2 -14852.48} C_VEL
LIN {X 0,Y 324.981,Z 480.667,A -85,B 0,C 180,E1 -14853.72,E2 -14853.72} C_VEL
LIN {X 0,Y 325.085,Z 478.92,A -85,B 0,C 180,E1 -14854.961,E2 -14854.961} C_VEL
LIN {X 0,Y 325.362,Z 475.279,A -85,B 0,C 180,E1 -14856.761,E2 -14856.761} C_VEL
LIN {X 0,Y 325.877,Z 469.958,A -85,B 0,C 180,E1 -14858.683,E2 -14858.683} C_VEL
LIN {X 0,Y 326.658,Z 463.142,A -85,B 0,C 180,E1 -14860.537,E2 -14860.537} C_VEL
LIN {X 0,Y 327.498,Z 455.689,A -85,B 0,C 180,E1 -14862.077,E2 -14862.077} C_VEL
LIN {X 0,Y 328.331,Z 448.337,A -85,B 0,C 180,E1 -14863.303,E2 -14863.303} C_VEL
LIN {X 0,Y 329.134,Z 440.46,A -85,B 0,C 180,E1 -14864.372,E2 -14864.372} C_VEL
LIN {X 0,Y 330.001,Z 432.133,A -85,B 0,C 180,E1 -14865.28,E2 -14865.28} C_VEL
LIN {X 0,Y 330.854,Z 421.488,A -85,B 0,C 180,E1 -14866.188,E2 -14866.188} C_VEL
LIN {X 0,Y 331.538,Z 409.88,A -85,B 0,C 180,E1 -14866.866,E2 -14866.866} C_VEL
LIN {X 0,Y 331.915,Z 401.43,A -85,B 0,C 180,E1 -14867.204,E2 -14867.204} C_VEL
LIN {X 0,Y 332.363,Z 375.032,A -85,B 0,C 180,E1 -14867.813,E2 -14867.813} C_VEL
LIN {X 0,Y 332.625,Z 351.254,A -85,B 0,C 180,E1 -14868.328,E2 -14868.328} C_VEL
LIN {X 0,Y 328.128,Z 325.037,A -85,B 0,C 180,E1 -14869.191,E2 -14869.191} C_VEL
LIN {X 0,Y 327.946,Z 323.561,A -85,B 0,C 180,E1 -14869.32,E2 -14869.32} C_VEL
LIN {X 0,Y 328.478,Z 317.29,A -85,B 0,C 180,E1 -14871.329,E2 -14871.329} C_VEL
LIN {X 0,Y 328.145,Z 312.622,A -85,B 0,C 180,E1 -14872.935,E2 -14872.935} C_VEL
LIN {X 0,Y 326.662,Z 304.71,A -85,B 0,C 180,E1 -14875.827,E2 -14875.827} C_VEL
LIN {X 0,Y 326.613,Z 304.613,A -85,B 0,C 180,E1 -14879.663,E2 -14879.663} C_VEL
LIN {X 0,Y 326.614,Z 304.613,A -85,B 0,C 180,E1 -14882.945,E2 -14882.945} C_VEL
LIN {X 0,Y 326.608,Z 304.613,A -85,B 0,C 180,E1 -14885.519,E2 -14885.519} C_VEL
LIN {X 0,Y 326.583,Z 304.617,A -85,B 0,C 180,E1 -14889.221,E2 -14889.221} C_VEL
LIN {X 0,Y 326.566,Z 304.615,A -85,B 0,C 180,E1 -14892.97,E2 -14892.97} C_VEL
LIN {X 0,Y 326.566,Z 304.62,A -85,B 0,C 180,E1 -14897.029,E2 -14897.029} C_VEL
LIN {X 0,Y 326.565,Z 304.609,A -85,B 0,C 180,E1 -14900.781,E2 -14900.781} C_VEL
LIN {X 0,Y 326.604,Z 304.611,A -85,B 0,C 180,E1 -14904.479,E2 -14904.479} C_VEL
LIN {X 0,Y 326.601,Z 304.612,A -85,B 0,C 180,E1 -14907.455,E2 -14907.455} C_VEL
LIN {X 0,Y 326.608,Z 304.61,A -85,B 0,C 180,E1 -14910.336,E2 -14910.336} C_VEL
LIN {X 0,Y 326.593,Z 304.617,A -85,B 0,C 180,E1 -14914.508,E2 -14914.508} C_VEL
LIN {X 0,Y 326.6,Z 304.613,A -85,B 0,C 180,E1 -14918.542,E2 -14918.542} C_VEL
LIN {X 0,Y 326.623,Z 304.614,A -85,B 0,C 180,E1 -14922.468,E2 -14922.468} C_VEL
LIN {X 0,Y 326.735,Z 304.595,A -85,B 0,C 180,E1 -14926.314,E2 -14926.314} C_VEL
LIN {X 0,Y 326.775,Z 304.593,A -85,B 0,C 180,E1 -14930.093,E2 -14930.093} C_VEL
LIN {X 0,Y 326.933,Z 304.571,A -85,B 0,C 180,E1 -14933.83,E2 -14933.83} C_VEL
LIN {X 0,Y 326.999,Z 304.561,A -85,B 0,C 180,E1 -14937.537,E2 -14937.537} C_VEL
LIN {X 0,Y 327.018,Z 304.56,A -85,B 0,C 180,E1 -14941.232,E2 -14941.232} C_VEL
LIN {X 0,Y 326.728,Z 304.597,A -85,B 0,C 180,E1 -14943.7,E2 -14943.7} C_VEL
LIN {X 0,Y 326.913,Z 304.572,A -85,B 0,C 180,E1 -14946.444,E2 -14946.444} C_VEL
LIN {X 0,Y 326.773,Z 304.594,A -85,B 0,C 180,E1 -14949.908,E2 -14949.908} C_VEL
LIN {X 0,Y 326.734,Z 304.595,A -85,B 0,C 180,E1 -14953.687,E2 -14953.687} C_VEL
LIN {X 0,Y 326.623,Z 304.613,A -85,B 0,C 180,E1 -14957.532,E2 -14957.532} C_VEL
LIN {X 0,Y 326.601,Z 304.613,A -85,B 0,C 180,E1 -14961.458,E2 -14961.458} C_VEL
LIN {X 0,Y 326.592,Z 304.618,A -85,B 0,C 180,E1 -14965.492,E2 -14965.492} C_VEL
LIN {X 0,Y 326.607,Z 304.611,A -85,B 0,C 180,E1 -14969.665,E2 -14969.665} C_VEL
LIN {X 0,Y 326.611,Z 304.613,A -85,B 0,C 180,E1 -14972.946,E2 -14972.946} C_VEL
LIN {X 0,Y 326.605,Z 304.611,A -85,B 0,C 180,E1 -14975.521,E2 -14975.521} C_VEL
LIN {X 0,Y 326.566,Z 304.609,A -85,B 0,C 180,E1 -14979.219,E2 -14979.219} C_VEL
LIN {X 0,Y 326.567,Z 304.62,A -85,B 0,C 180,E1 -14982.972,E2 -14982.972} C_VEL
LIN {X 0,Y 326.567,Z 304.615,A -85,B 0,C 180,E1 -14987.03,E2 -14987.03} C_VEL
LIN {X 0,Y 326.579,Z 304.616,A -85,B 0,C 180,E1 -14991.386,E2 -14991.386} C_VEL
LIN {X 0,Y 326.616,Z 304.61,A -85,B 0,C 180,E1 -14994.852,E2 -14994.852} C_VEL
LIN {X 0,Y 326.606,Z 304.612,A -85,B 0,C 180,E1 -14997.456,E2 -14997.456} C_VEL
LIN {X 0,Y 326.578,Z 304.618,A -85,B 0,C 180,E1 -15000.333,E2 -15000.333} C_VEL
LIN {X 0,Y 326.686,Z 304.775,A -85,B 0,C 180,E1 -15004.26,E2 -15004.26} C_VEL
LIN {X 0,Y 328.259,Z 313.254,A -85,B 0,C 180,E1 -15007.333,E2 -15007.333} C_VEL
LIN {X 0,Y 328.476,Z 317.157,A -85,B 0,C 180,E1 -15008.671,E2 -15008.671} C_VEL
LIN {X 0,Y 327.942,Z 323.741,A -85,B 0,C 180,E1 -15010.762,E2 -15010.762} C_VEL
LIN {X 0,Y 328.846,Z 328.655,A -85,B 0,C 180,E1 -15010.989,E2 -15010.989} C_VEL
LIN {X 0,Y 332.716,Z 352.078,A -85,B 0,C 180,E1 -15011.741,E2 -15011.741} C_VEL
LIN {X 0,Y 331.963,Z 399.959,A -85,B 0,C 180,E1 -15012.799,E2 -15012.799} C_VEL
LIN {X 0,Y 331.557,Z 409.768,A -85,B 0,C 180,E1 -15013.174,E2 -15013.174} C_VEL
LIN {X 0,Y 330.896,Z 420.874,A -85,B 0,C 180,E1 -15013.814,E2 -15013.814} C_VEL
LIN {X 0,Y 330.037,Z 431.706,A -85,B 0,C 180,E1 -15014.721,E2 -15014.721} C_VEL
LIN {X 0,Y 329.21,Z 440.11,A -85,B 0,C 180,E1 -15015.631,E2 -15015.631} C_VEL
LIN {X 0,Y 328.355,Z 448.045,A -85,B 0,C 180,E1 -15016.698,E2 -15016.698} C_VEL
LIN {X 0,Y 327.762,Z 453.744,A -85,B 0,C 180,E1 -15017.619,E2 -15017.619} C_VEL
LIN {X 0,Y 326.986,Z 460.109,A -85,B 0,C 180,E1 -15018.847,E2 -15018.847} C_VEL
LIN {X 0,Y 326.258,Z 466.574,A -85,B 0,C 180,E1 -15020.39,E2 -15020.39} C_VEL
LIN {X 0,Y 325.727,Z 471.733,A -85,B 0,C 180,E1 -15021.938,E2 -15021.938} C_VEL
LIN {X 0,Y 325.233,Z 476.507,A -85,B 0,C 180,E1 -15023.797,E2 -15023.797} C_VEL
LIN {X 0,Y 325.099,Z 478.837,A -85,B 0,C 180,E1 -15025.039,E2 -15025.039} C_VEL
LIN {X 0,Y 324.986,Z 480.608,A -85,B 0,C 180,E1 -15026.28,E2 -15026.28} C_VEL
LIN {X 0,Y 324.847,Z 481.885,A -85,B 0,C 180,E1 -15027.52,E2 -15027.52} C_VEL
LIN {X 0,Y 324.787,Z 482.691,A -85,B 0,C 180,E1 -15028.76,E2 -15028.76} C_VEL
LIN {X 0,Y 324.766,Z 482.998,A -85,B 0,C 180,E1 -15030,E2 -15030} C_VEL
LIN {X 0,Y 324.783,Z 482.719,A -85,B 0,C 180,E1 -15031.24,E2 -15031.24} C_VEL
LIN {X 0,Y 324.836,Z 481.97,A -85,B 0,C 180,E1 -15032.48,E2 -15032.48} C_VEL
LIN {X 0,Y 324.956,Z 480.75,A -85,B 0,C 180,E1 -15033.72,E2 -15033.72} C_VEL
LIN {X 0,Y 325.082,Z 479.038,A -85,B 0,C 180,E1 -15034.961,E2 -15034.961} C_VEL
LIN {X 0,Y 325.353,Z 475.433,A -85,B 0,C 180,E1 -15036.761,E2 -15036.761} C_VEL
LIN {X 0,Y 325.872,Z 470.155,A -85,B 0,C 180,E1 -15038.683,E2 -15038.683} C_VEL
LIN {X 0,Y 326.477,Z 464.641,A -85,B 0,C 180,E1 -15040.23,E2 -15040.23} C_VEL
LIN {X 0,Y 327.347,Z 457.716,A -85,B 0,C 180,E1 -15041.768,E2 -15041.768} C_VEL
LIN {X 0,Y 328.19,Z 449.765,A -85,B 0,C 180,E1 -15043.151,E2 -15043.151} C_VEL
LIN {X 0,Y 328.977,Z 442.186,A -85,B 0,C 180,E1 -15044.221,E2 -15044.221} C_VEL
LIN {X 0,Y 329.842,Z 434.242,A -85,B 0,C 180,E1 -15045.13,E2 -15045.13} C_VEL
LIN {X 0,Y 330.563,Z 426.038,A -85,B 0,C 180,E1 -15045.886,E2 -15045.886} C_VEL
LIN {X 0,Y 331.173,Z 417.722,A -85,B 0,C 180,E1 -15046.489,E2 -15046.489} C_VEL
LIN {X 0,Y 331.622,Z 408.733,A -85,B 0,C 180,E1 -15046.981,E2 -15046.981} C_VEL
LIN {X 0,Y 332.023,Z 399.149,A -85,B 0,C 180,E1 -15047.332,E2 -15047.332} C_VEL
LIN {X 0,Y 332.693,Z 351.706,A -85,B 0,C 180,E1 -15048.378,E2 -15048.378} C_VEL
LIN {X 0,Y 328.627,Z 327.541,A -85,B 0,C 180,E1 -15049.16,E2 -15049.16} C_VEL
LIN {X 0,Y 327.952,Z 323.647,A -85,B 0,C 180,E1 -15049.361,E2 -15049.361} C_VEL
LIN {X 0,Y 328.472,Z 317.487,A -85,B 0,C 180,E1 -15051.329,E2 -15051.329} C_VEL
LIN {X 0,Y 328.16,Z 312.799,A -85,B 0,C 180,E1 -15052.941,E2 -15052.941} C_VEL
LIN {X 0,Y 326.667,Z 304.695,A -85,B 0,C 180,E1 -15055.912,E2 -15055.912} C_VEL
LIN {X 0,Y 326.614,Z 304.614,A -85,B 0,C 180,E1 -15059.663,E2 -15059.663} C_VEL
LIN {X 0,Y 326.615,Z 304.612,A -85,B 0,C 180,E1 -15062.945,E2 -15062.945} C_VEL
LIN {X 0,Y 326.596,Z 304.612,A -85,B 0,C 180,E1 -15065.773,E2 -15065.773} C_VEL
LIN {X 0,Y 325.892,Z 304.702,A -85,B 0,C 180,E1 -15066.801,E2 -15066.801} C_VEL
LIN {X 0,Y 322.985,Z 305.063,A -85,B 0,C 180,E1 -15068.474,E2 -15068.474} C_VEL
LIN {X 0,Y 320.561,Z 305.361,A -85,B 0,C 180,E1 -15069.829,E2 -15069.829} C_VEL
LIN {X 0,Y 319.555,Z 305.487,A -85,B 0,C 180,E1 -15070.88,E2 -15070.88} C_VEL
LIN {X 0,Y 319.491,Z 305.492,A -85,B 0,C 180,E1 -15071.235,E2 -15071.235} C_VEL
